Yaskawa INFORM job: A_ROOF_SIDE_0617_2_PAINT_9.JBI

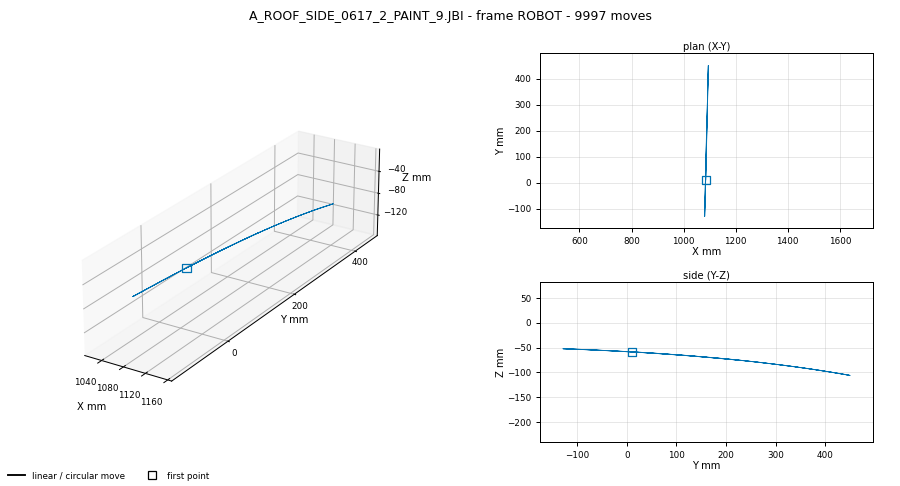
[picture p0: tool path of A_ROOF_SIDE_0617_2_PAINT_9.JBI in frame ROBOT, 9997 of 9997 moves have a stored position in this frame; points joined in program order, loops and branches not executed]
/JOB
//NAME A_ROOF_SIDE_0617_2_PAINT9
//POS
///NPOS 9997,0,0,0,0,0
///TOOL 1
///USER 0
///POSTYPE ROBOT
///RECTAN
///RCONF 1,0,0,0,0,0,0,0,0,0,0,0,0,0,0,0,0,0,0,0,0,0,0,0
C00000=1085.245,10.844,-58.197,174.491,19.105,153.128
C00001=1085.250,11.093,-58.211,174.492,19.107,153.129
C00002=1085.256,11.342,-58.226,174.493,19.109,153.129
C00003=1085.262,11.592,-58.240,174.496,19.111,153.129
C00004=1085.269,11.841,-58.254,174.497,19.113,153.129
C00005=1085.275,12.091,-58.268,174.498,19.115,153.129
C00006=1085.280,12.340,-58.283,174.500,19.118,153.129
C00007=1085.286,12.590,-58.297,174.502,19.119,153.129
C00008=1085.292,12.839,-58.312,174.503,19.121,153.129
C00009=1085.298,13.089,-58.325,174.505,19.123,153.129
C00010=1085.304,13.338,-58.340,174.507,19.125,153.130
C00011=1085.310,13.588,-58.354,174.508,19.127,153.130
C00012=1085.315,13.837,-58.369,174.509,19.129,153.130
C00013=1085.321,14.087,-58.383,174.512,19.131,153.130
C00014=1085.327,14.336,-58.398,174.513,19.133,153.130
C00015=1085.333,14.586,-58.412,174.514,19.134,153.130
C00016=1085.340,14.863,-58.428,174.516,19.137,153.130
C00017=1085.346,15.140,-58.445,174.517,19.139,153.130
C00018=1085.352,15.417,-58.461,174.520,19.141,153.130
C00019=1085.358,15.693,-58.476,174.521,19.143,153.131
C00020=1085.365,15.943,-58.491,174.523,19.145,153.131
C00021=1085.370,16.192,-58.505,174.524,19.147,153.131
C00022=1085.376,16.443,-58.520,174.526,19.149,153.131
C00023=1085.382,16.692,-58.535,174.528,19.151,153.131
C00024=1085.387,16.941,-58.549,174.529,19.153,153.131
C00025=1085.393,17.191,-58.564,174.530,19.155,153.131
C00026=1085.399,17.440,-58.578,174.533,19.157,153.131
C00027=1085.405,17.689,-58.592,174.534,19.159,153.131
C00028=1085.411,17.939,-58.607,174.535,19.161,153.132
C00029=1085.416,18.188,-58.622,174.537,19.163,153.132
C00030=1085.422,18.438,-58.636,174.539,19.165,153.132
C00031=1085.428,18.687,-58.651,174.540,19.167,153.132
C00032=1085.434,18.937,-58.666,174.541,19.168,153.132
C00033=1085.440,19.187,-58.680,174.544,19.171,153.132
C00034=1085.445,19.436,-58.695,174.545,19.173,153.132
C00035=1085.451,19.686,-58.710,174.546,19.174,153.132
C00036=1085.457,19.935,-58.724,174.548,19.177,153.132
C00037=1085.463,20.185,-58.739,174.550,19.178,153.132
C00038=1085.469,20.434,-58.753,174.551,19.181,153.133
C00039=1085.474,20.684,-58.769,174.553,19.183,153.133
C00040=1085.480,20.933,-58.783,174.554,19.185,153.133
C00041=1085.486,21.182,-58.797,174.556,19.186,153.133
C00042=1085.491,21.432,-58.813,174.558,19.189,153.133
C00043=1085.497,21.681,-58.827,174.559,19.191,153.133
C00044=1085.503,21.931,-58.842,174.561,19.192,153.133
C00045=1085.509,22.180,-58.856,174.563,19.195,153.133
C00046=1085.515,22.430,-58.872,174.564,19.196,153.133
C00047=1085.520,22.679,-58.886,174.565,19.198,153.134
C00048=1085.527,22.930,-58.901,174.568,19.200,153.134
C00049=1085.532,23.179,-58.916,174.569,19.202,153.134
C00050=1085.538,23.429,-58.931,174.570,19.204,153.134
C00051=1085.544,23.677,-58.945,174.572,19.206,153.134
C00052=1085.549,23.927,-58.960,174.574,19.208,153.134
C00053=1085.555,24.176,-58.975,174.575,19.210,153.134
C00054=1085.561,24.426,-58.989,174.577,19.212,153.134
C00055=1085.566,24.676,-59.005,174.578,19.214,153.134
C00056=1085.572,24.925,-59.019,174.580,19.216,153.135
C00057=1085.578,25.175,-59.034,174.582,19.218,153.135
C00058=1085.584,25.424,-59.049,174.583,19.220,153.135
C00059=1085.590,25.674,-59.064,174.585,19.222,153.135
C00060=1085.596,25.922,-59.079,174.587,19.224,153.135
C00061=1085.601,26.172,-59.095,174.588,19.226,153.135
C00062=1085.607,26.421,-59.109,174.589,19.228,153.135
C00063=1085.613,26.672,-59.123,174.592,19.230,153.135
C00064=1085.619,26.922,-59.139,174.593,19.232,153.135
C00065=1085.625,27.171,-59.153,174.594,19.233,153.135
C00066=1085.630,27.421,-59.169,174.596,19.236,153.136
C00067=1085.636,27.670,-59.184,174.598,19.237,153.136
C00068=1085.642,27.919,-59.199,174.599,19.239,153.136
C00069=1085.647,28.168,-59.214,174.601,19.241,153.136
C00070=1085.654,28.418,-59.229,174.602,19.243,153.136
C00071=1085.659,28.667,-59.244,174.604,19.245,153.136
C00072=1085.665,28.917,-59.259,174.606,19.247,153.136
C00073=1085.670,29.166,-59.274,174.607,19.249,153.136
C00074=1085.677,29.416,-59.289,174.609,19.251,153.136
C00075=1085.682,29.665,-59.304,174.611,19.253,153.137
C00076=1085.688,29.915,-59.319,174.612,19.255,153.137
C00077=1085.693,30.164,-59.334,174.613,19.257,153.137
C00078=1085.700,30.414,-59.349,174.616,19.259,153.137
C00079=1085.705,30.664,-59.365,174.617,19.261,153.137
C00080=1085.712,30.942,-59.382,174.619,19.263,153.137
C00081=1085.718,31.220,-59.398,174.620,19.265,153.137
C00082=1085.725,31.498,-59.415,174.622,19.268,153.137
C00083=1085.731,31.776,-59.432,174.624,19.270,153.137
C00084=1085.736,32.025,-59.447,174.626,19.272,153.137
C00085=1085.743,32.275,-59.462,174.627,19.274,153.138
C00086=1085.748,32.525,-59.478,174.629,19.276,153.138
C00087=1085.754,32.774,-59.493,174.631,19.278,153.138
C00088=1085.760,33.023,-59.508,174.632,19.279,153.138
C00089=1085.765,33.273,-59.524,174.634,19.282,153.138
C00090=1085.771,33.522,-59.538,174.636,19.283,153.138
C00091=1085.776,33.772,-59.554,174.637,19.285,153.138
C00092=1085.783,34.021,-59.569,174.639,19.287,153.138
C00093=1085.788,34.271,-59.584,174.640,19.289,153.138
C00094=1085.794,34.520,-59.600,174.643,19.291,153.138
C00095=1085.800,34.770,-59.615,174.644,19.293,153.139
C00096=1085.806,35.020,-59.630,174.645,19.295,153.139
C00097=1085.812,35.268,-59.645,174.647,19.298,153.139
C00098=1085.817,35.518,-59.661,174.649,19.299,153.139
C00099=1085.822,35.768,-59.676,174.650,19.301,153.139
C00100=1085.829,36.017,-59.691,174.652,19.303,153.139
C00101=1085.835,36.267,-59.707,174.654,19.305,153.139
C00102=1085.840,36.516,-59.722,174.655,19.307,153.139
C00103=1085.846,36.766,-59.737,174.657,19.309,153.139
C00104=1085.852,37.015,-59.753,174.659,19.311,153.139
C00105=1085.858,37.264,-59.768,174.661,19.313,153.139
C00106=1085.863,37.514,-59.783,174.662,19.315,153.140
C00107=1085.870,37.764,-59.798,174.663,19.316,153.140
C00108=1085.875,38.012,-59.814,174.666,19.319,153.140
C00109=1085.881,38.262,-59.830,174.667,19.320,153.140
C00110=1085.886,38.512,-59.845,174.668,19.322,153.140
C00111=1085.893,38.760,-59.861,174.671,19.324,153.140
C00112=1085.898,39.010,-59.876,174.672,19.326,153.140
C00113=1085.904,39.260,-59.892,174.674,19.328,153.140
C00114=1085.909,39.509,-59.908,174.675,19.330,153.140
C00115=1085.915,39.759,-59.923,174.677,19.332,153.140
C00116=1085.921,40.009,-59.938,174.679,19.334,153.141
C00117=1085.927,40.257,-59.954,174.680,19.336,153.141
C00118=1085.932,40.507,-59.970,174.682,19.338,153.141
C00119=1085.938,40.757,-59.985,174.684,19.340,153.141
C00120=1085.944,41.006,-60.000,174.685,19.342,153.141
C00121=1085.950,41.256,-60.016,174.687,19.344,153.141
C00122=1085.955,41.506,-60.032,174.688,19.346,153.141
C00123=1085.961,41.754,-60.047,174.690,19.348,153.141
C00124=1085.966,42.004,-60.063,174.692,19.350,153.141
C00125=1085.972,42.253,-60.079,174.693,19.352,153.141
C00126=1085.978,42.502,-60.094,174.695,19.354,153.142
C00127=1085.984,42.752,-60.110,174.697,19.356,153.142
C00128=1085.990,43.002,-60.126,174.698,19.357,153.142
C00129=1085.995,43.252,-60.141,174.700,19.360,153.142
C00130=1086.001,43.500,-60.157,174.702,19.361,153.142
C00131=1086.007,43.750,-60.172,174.704,19.364,153.142
C00132=1086.013,43.999,-60.188,174.705,19.365,153.142
C00133=1086.018,44.249,-60.203,174.707,19.367,153.142
C00134=1086.024,44.498,-60.220,174.709,19.369,153.142
C00135=1086.030,44.748,-60.235,174.710,19.371,153.142
C00136=1086.035,44.997,-60.251,174.712,19.373,153.142
C00137=1086.041,45.247,-60.267,174.714,19.375,153.143
C00138=1086.047,45.496,-60.283,174.715,19.377,153.143
C00139=1086.052,45.746,-60.298,174.717,19.379,153.143
C00140=1086.058,45.995,-60.314,174.719,19.381,153.143
C00141=1086.063,46.245,-60.330,174.721,19.383,153.143
C00142=1086.069,46.494,-60.346,174.722,19.385,153.143
C00143=1086.074,46.743,-60.361,174.723,19.387,153.143
C00144=1086.081,47.022,-60.379,174.726,19.389,153.143
C00145=1086.087,47.300,-60.397,174.728,19.391,153.143
C00146=1086.092,47.578,-60.415,174.729,19.393,153.144
C00147=1086.100,47.857,-60.432,174.731,19.396,153.144
C00148=1086.105,48.105,-60.448,174.733,19.398,153.144
C00149=1086.111,48.355,-60.465,174.735,19.400,153.144
C00150=1086.117,48.605,-60.480,174.736,19.402,153.144
C00151=1086.123,48.854,-60.496,174.738,19.404,153.144
C00152=1086.127,49.103,-60.513,174.740,19.406,153.144
C00153=1086.133,49.353,-60.528,174.742,19.408,153.144
C00154=1086.139,49.602,-60.545,174.743,19.410,153.144
C00155=1086.144,49.852,-60.560,174.745,19.411,153.144
C00156=1086.150,50.102,-60.576,174.747,19.413,153.144
C00157=1086.156,50.350,-60.592,174.748,19.415,153.145
C00158=1086.161,50.600,-60.608,174.750,19.417,153.145
C00159=1086.167,50.850,-60.624,174.752,19.419,153.145
C00160=1086.173,51.099,-60.640,174.753,19.421,153.145
C00161=1086.179,51.348,-60.657,174.755,19.423,153.145
C00162=1086.184,51.598,-60.672,174.757,19.425,153.145
C00163=1086.190,51.847,-60.688,174.759,19.427,153.145
C00164=1086.196,52.096,-60.704,174.760,19.429,153.145
C00165=1086.202,52.346,-60.721,174.762,19.431,153.145
C00166=1086.207,52.596,-60.737,174.764,19.433,153.145
C00167=1086.212,52.845,-60.753,174.765,19.434,153.145
C00168=1086.218,53.094,-60.769,174.767,19.436,153.145
C00169=1086.224,53.343,-60.785,174.769,19.438,153.146
C00170=1086.230,53.593,-60.801,174.771,19.440,153.146
C00171=1086.236,53.843,-60.817,174.772,19.442,153.146
C00172=1086.242,54.092,-60.833,174.774,19.444,153.146
C00173=1086.248,54.341,-60.849,174.776,19.446,153.146
C00174=1086.253,54.590,-60.865,174.777,19.447,153.146
C00175=1086.258,54.840,-60.881,174.779,19.450,153.146
C00176=1086.264,55.089,-60.898,174.781,19.451,153.146
C00177=1086.270,55.339,-60.914,174.783,19.454,153.146
C00178=1086.276,55.588,-60.930,174.784,19.455,153.146
C00179=1086.282,55.838,-60.946,174.787,19.457,153.146
C00180=1086.288,56.087,-60.963,174.788,19.460,153.146
C00181=1086.293,56.337,-60.978,174.789,19.461,153.146
C00182=1086.299,56.587,-60.995,174.792,19.463,153.146
C00183=1086.305,56.836,-61.011,174.793,19.465,153.146
C00184=1086.310,57.085,-61.027,174.795,19.467,153.147
C00185=1086.316,57.334,-61.044,174.797,19.469,153.147
C00186=1086.322,57.583,-61.060,174.799,19.471,153.147
C00187=1086.328,57.833,-61.076,174.800,19.473,153.147
C00188=1086.333,58.082,-61.093,174.802,19.474,153.147
C00189=1086.339,58.332,-61.109,174.804,19.476,153.147
C00190=1086.345,58.581,-61.125,174.805,19.478,153.147
C00191=1086.351,58.830,-61.142,174.808,19.480,153.147
C00192=1086.357,59.080,-61.158,174.809,19.482,153.147
C00193=1086.362,59.329,-61.175,174.811,19.484,153.147
C00194=1086.368,59.579,-61.191,174.813,19.486,153.147
C00195=1086.374,59.828,-61.207,174.814,19.487,153.147
C00196=1086.380,60.077,-61.224,174.816,19.489,153.147
C00197=1086.386,60.327,-61.240,174.818,19.491,153.147
C00198=1086.391,60.576,-61.257,174.820,19.493,153.148
C00199=1086.397,60.826,-61.273,174.821,19.495,153.148
C00200=1086.403,61.075,-61.289,174.824,19.497,153.148
C00201=1086.409,61.324,-61.305,174.825,19.498,153.148
C00202=1086.415,61.574,-61.322,174.827,19.501,153.148
C00203=1086.420,61.823,-61.339,174.829,19.502,153.148
C00204=1086.426,62.073,-61.355,174.830,19.504,153.148
C00205=1086.432,62.322,-61.371,174.832,19.506,153.148
C00206=1086.438,62.571,-61.387,174.834,19.507,153.148
C00207=1086.443,62.821,-61.404,174.836,19.510,153.148
C00208=1086.451,63.099,-61.422,174.838,19.512,153.148
C00209=1086.457,63.376,-61.441,174.840,19.513,153.148
C00210=1086.463,63.655,-61.459,174.842,19.516,153.148
C00211=1086.470,63.933,-61.477,174.844,19.518,153.148
C00212=1086.476,64.182,-61.494,174.845,19.519,153.148
C00213=1086.481,64.432,-61.511,174.848,19.521,153.148
C00214=1086.487,64.681,-61.527,174.849,19.523,153.149
C00215=1086.492,64.930,-61.544,174.851,19.525,153.149
C00216=1086.498,65.180,-61.561,174.853,19.527,153.149
C00217=1086.504,65.429,-61.577,174.855,19.529,153.149
C00218=1086.509,65.679,-61.594,174.856,19.531,153.149
C00219=1086.515,65.928,-61.610,174.858,19.532,153.149
C00220=1086.521,66.177,-61.628,174.860,19.534,153.149
C00221=1086.527,66.426,-61.644,174.862,19.536,153.149
C00222=1086.532,66.676,-61.661,174.864,19.538,153.149
C00223=1086.538,66.925,-61.677,174.865,19.540,153.149
C00224=1086.544,67.175,-61.693,174.867,19.542,153.149
C00225=1086.550,67.424,-61.711,174.869,19.543,153.149
C00226=1086.556,67.674,-61.727,174.871,19.545,153.149
C00227=1086.561,67.923,-61.744,174.872,19.547,153.149
C00228=1086.567,68.173,-61.760,174.875,19.549,153.149
C00229=1086.573,68.422,-61.778,174.876,19.551,153.149
C00230=1086.579,68.671,-61.794,174.878,19.553,153.149
C00231=1086.584,68.921,-61.811,174.880,19.554,153.149
C00232=1086.590,69.170,-61.828,174.882,19.557,153.150
C00233=1086.595,69.419,-61.845,174.883,19.558,153.150
C00234=1086.601,69.669,-61.861,174.885,19.560,153.150
C00235=1086.607,69.918,-61.879,174.887,19.562,153.150
C00236=1086.612,70.167,-61.896,174.889,19.564,153.150
C00237=1086.618,70.417,-61.912,174.891,19.566,153.150
C00238=1086.624,70.666,-61.929,174.892,19.568,153.150
C00239=1086.629,70.915,-61.946,174.895,19.570,153.150
C00240=1086.635,71.165,-61.963,174.896,19.571,153.150
C00241=1086.641,71.414,-61.980,174.898,19.573,153.150
C00242=1086.647,71.664,-61.997,174.900,19.575,153.150
C00243=1086.652,71.913,-62.014,174.902,19.577,153.150
C00244=1086.658,72.162,-62.031,174.903,19.579,153.150
C00245=1086.663,72.412,-62.047,174.906,19.581,153.150
C00246=1086.669,72.661,-62.065,174.907,19.582,153.150
C00247=1086.675,72.910,-62.081,174.909,19.585,153.150
C00248=1086.680,73.159,-62.099,174.911,19.586,153.150
C00249=1086.686,73.409,-62.116,174.913,19.588,153.150
C00250=1086.692,73.658,-62.133,174.914,19.590,153.151
C00251=1086.698,73.908,-62.150,174.917,19.592,153.151
C00252=1086.703,74.158,-62.167,174.918,19.593,153.151
C00253=1086.709,74.406,-62.184,174.921,19.595,153.151
C00254=1086.714,74.656,-62.201,174.922,19.597,153.151
C00255=1086.720,74.905,-62.218,174.924,19.599,153.151
C00256=1086.726,75.154,-62.234,174.926,19.601,153.151
C00257=1086.732,75.404,-62.252,174.928,19.603,153.151
C00258=1086.737,75.654,-62.269,174.929,19.604,153.151
C00259=1086.743,75.902,-62.286,174.932,19.606,153.151
C00260=1086.749,76.152,-62.304,174.933,19.608,153.151
C00261=1086.754,76.401,-62.321,174.935,19.610,153.151
C00262=1086.760,76.650,-62.337,174.937,19.612,153.151
C00263=1086.766,76.900,-62.355,174.939,19.614,153.151
C00264=1086.772,77.149,-62.372,174.940,19.615,153.151
C00265=1086.777,77.399,-62.389,174.943,19.617,153.151
C00266=1086.783,77.648,-62.406,174.944,19.619,153.151
C00267=1086.789,77.897,-62.424,174.947,19.621,153.151
C00268=1086.795,78.147,-62.441,174.948,19.622,153.151
C00269=1086.800,78.396,-62.458,174.950,19.624,153.151
C00270=1086.806,78.646,-62.475,174.952,19.626,153.151
C00271=1086.812,78.895,-62.492,174.954,19.628,153.151
C00272=1086.818,79.173,-62.512,174.956,19.630,153.151
C00273=1086.824,79.450,-62.531,174.958,19.632,153.152
C00274=1086.830,79.728,-62.550,174.960,19.634,153.152
C00275=1086.836,80.007,-62.570,174.962,19.636,153.152
C00276=1086.843,80.256,-62.587,174.964,19.637,153.152
C00277=1086.848,80.505,-62.604,174.966,19.640,153.152
C00278=1086.853,80.754,-62.621,174.967,19.641,153.152
C00279=1086.859,81.003,-62.639,174.970,19.643,153.152
C00280=1086.865,81.253,-62.657,174.972,19.645,153.152
C00281=1086.870,81.503,-62.673,174.973,19.647,153.152
C00282=1086.876,81.752,-62.691,174.976,19.649,153.152
C00283=1086.881,82.001,-62.709,174.977,19.650,153.152
C00284=1086.887,82.251,-62.727,174.979,19.652,153.152
C00285=1086.893,82.500,-62.743,174.981,19.654,153.152
C00286=1086.898,82.749,-62.761,174.983,19.656,153.152
C00287=1086.904,82.998,-62.778,174.985,19.657,153.152
C00288=1086.910,83.247,-62.795,174.987,19.659,153.152
C00289=1086.916,83.497,-62.813,174.988,19.661,153.152
C00290=1086.921,83.747,-62.830,174.991,19.663,153.152
C00291=1086.927,83.996,-62.848,174.992,19.665,153.152
C00292=1086.933,84.245,-62.866,174.994,19.667,153.152
C00293=1086.938,84.494,-62.883,174.996,19.668,153.152
C00294=1086.944,84.743,-62.901,174.998,19.670,153.152
C00295=1086.949,84.992,-62.918,175.000,19.672,153.152
C00296=1086.955,85.243,-62.936,175.002,19.674,153.152
C00297=1086.961,85.492,-62.953,175.003,19.675,153.152
C00298=1086.966,85.741,-62.971,175.006,19.677,153.152
C00299=1086.972,85.990,-62.988,175.007,19.679,153.152
C00300=1086.978,86.240,-63.006,175.009,19.681,153.152
C00301=1086.983,86.489,-63.024,175.012,19.683,153.152
C00302=1086.989,86.738,-63.041,175.013,19.684,153.153
C00303=1086.995,86.987,-63.059,175.016,19.686,153.152
C00304=1087.000,87.237,-63.076,175.017,19.687,153.152
C00305=1087.006,87.486,-63.094,175.020,19.689,153.152
C00306=1087.012,87.736,-63.112,175.021,19.691,153.153
C00307=1087.017,87.985,-63.129,175.023,19.693,153.153
C00308=1087.023,88.234,-63.147,175.025,19.694,153.153
C00309=1087.029,88.484,-63.165,175.027,19.696,153.153
C00310=1087.035,88.733,-63.182,175.029,19.698,153.153
C00311=1087.040,88.982,-63.200,175.031,19.700,153.153
C00312=1087.046,89.232,-63.218,175.032,19.701,153.153
C00313=1087.052,89.481,-63.235,175.035,19.703,153.153
C00314=1087.058,89.730,-63.253,175.037,19.705,153.153
C00315=1087.063,89.979,-63.271,175.039,19.707,153.153
C00316=1087.069,90.228,-63.288,175.041,19.708,153.153
C00317=1087.075,90.478,-63.306,175.043,19.710,153.153
C00318=1087.080,90.727,-63.324,175.045,19.712,153.153
C00319=1087.087,90.977,-63.342,175.046,19.713,153.153
C00320=1087.092,91.226,-63.359,175.049,19.715,153.153
C00321=1087.097,91.475,-63.378,175.050,19.717,153.153
C00322=1087.103,91.724,-63.396,175.052,19.719,153.153
C00323=1087.109,91.973,-63.414,175.055,19.721,153.153
C00324=1087.114,92.223,-63.431,175.056,19.722,153.153
C00325=1087.120,92.472,-63.449,175.059,19.724,153.153
C00326=1087.125,92.722,-63.468,175.060,19.726,153.153
C00327=1087.131,92.971,-63.485,175.062,19.728,153.153
C00328=1087.137,93.220,-63.503,175.064,19.729,153.153
C00329=1087.142,93.469,-63.521,175.066,19.731,153.153
C00330=1087.148,93.718,-63.539,175.068,19.732,153.153
C00331=1087.154,93.968,-63.557,175.070,19.734,153.153
C00332=1087.159,94.217,-63.575,175.072,19.736,153.153
C00333=1087.165,94.467,-63.593,175.074,19.738,153.153
C00334=1087.170,94.716,-63.611,175.076,19.740,153.153
C00335=1087.176,94.965,-63.629,175.078,19.741,153.153
C00336=1087.182,95.243,-63.649,175.080,19.743,153.153
C00337=1087.188,95.521,-63.669,175.082,19.745,153.153
C00338=1087.195,95.799,-63.689,175.085,19.747,153.153
C00339=1087.202,96.077,-63.710,175.087,19.749,153.153
C00340=1087.206,96.327,-63.728,175.088,19.751,153.153
C00341=1087.212,96.576,-63.745,175.091,19.752,153.153
C00342=1087.218,96.825,-63.764,175.092,19.754,153.153
C00343=1087.224,97.074,-63.781,175.095,19.756,153.153
C00344=1087.229,97.324,-63.800,175.097,19.758,153.153
C00345=1087.235,97.572,-63.818,175.099,19.759,153.153
C00346=1087.241,97.822,-63.836,175.101,19.761,153.153
C00347=1087.246,98.071,-63.854,175.103,19.762,153.153
C00348=1087.252,98.321,-63.873,175.105,19.764,153.153
C00349=1087.258,98.570,-63.891,175.107,19.766,153.153
C00350=1087.263,98.820,-63.909,175.109,19.768,153.153
C00351=1087.269,99.068,-63.927,175.111,19.769,153.153
C00352=1087.275,99.318,-63.945,175.113,19.771,153.153
C00353=1087.281,99.567,-63.963,175.115,19.773,153.153
C00354=1087.287,99.816,-63.982,175.117,19.774,153.153
C00355=1087.292,100.065,-64.000,175.119,19.776,153.153
C00356=1087.298,100.315,-64.018,175.121,19.778,153.153
C00357=1087.303,100.564,-64.037,175.123,19.779,153.153
C00358=1087.309,100.814,-64.054,175.125,19.781,153.153
C00359=1087.314,101.062,-64.073,175.127,19.782,153.153
C00360=1087.321,101.312,-64.091,175.129,19.784,153.153
C00361=1087.326,101.561,-64.109,175.132,19.786,153.153
C00362=1087.332,101.811,-64.128,175.133,19.788,153.153
C00363=1087.337,102.060,-64.146,175.135,19.790,153.153
C00364=1087.343,102.309,-64.165,175.137,19.791,153.153
C00365=1087.349,102.558,-64.182,175.139,19.793,153.153
C00366=1087.354,102.807,-64.202,175.142,19.795,153.153
C00367=1087.360,103.057,-64.219,175.143,19.796,153.153
C00368=1087.365,103.306,-64.239,175.145,19.798,153.153
C00369=1087.371,103.555,-64.256,175.147,19.799,153.153
C00370=1087.377,103.804,-64.275,175.150,19.801,153.153
C00371=1087.381,104.054,-64.293,175.152,19.803,153.153
C00372=1087.388,104.303,-64.312,175.153,19.804,153.153
C00373=1087.393,104.552,-64.330,175.156,19.806,153.153
C00374=1087.399,104.801,-64.349,175.157,19.807,153.153
C00375=1087.404,105.051,-64.367,175.160,19.809,153.153
C00376=1087.410,105.300,-64.386,175.162,19.811,153.153
C00377=1087.416,105.549,-64.405,175.164,19.812,153.153
C00378=1087.421,105.798,-64.423,175.166,19.814,153.153
C00379=1087.427,106.048,-64.442,175.167,19.816,153.153
C00380=1087.432,106.297,-64.460,175.170,19.817,153.153
C00381=1087.438,106.546,-64.479,175.172,19.819,153.153
C00382=1087.444,106.796,-64.498,175.174,19.821,153.153
C00383=1087.450,107.045,-64.515,175.176,19.822,153.153
C00384=1087.455,107.294,-64.535,175.178,19.824,153.153
C00385=1087.461,107.543,-64.552,175.180,19.826,153.153
C00386=1087.466,107.793,-64.571,175.183,19.827,153.153
C00387=1087.472,108.042,-64.591,175.184,19.829,153.153
C00388=1087.478,108.291,-64.608,175.187,19.831,153.153
C00389=1087.483,108.540,-64.628,175.189,19.832,153.152
C00390=1087.489,108.789,-64.646,175.191,19.834,153.153
C00391=1087.495,109.038,-64.665,175.193,19.836,153.153
C00392=1087.500,109.288,-64.684,175.195,19.837,153.152
C00393=1087.506,109.537,-64.702,175.197,19.839,153.152
C00394=1087.512,109.786,-64.721,175.199,19.840,153.152
C00395=1087.518,110.036,-64.739,175.201,19.842,153.152
C00396=1087.523,110.285,-64.758,175.203,19.844,153.152
C00397=1087.529,110.534,-64.777,175.206,19.845,153.152
C00398=1087.535,110.783,-64.796,175.207,19.847,153.152
C00399=1087.540,111.033,-64.814,175.210,19.848,153.152
C00400=1087.546,111.311,-64.836,175.212,19.850,153.152
C00401=1087.553,111.589,-64.856,175.215,19.852,153.152
C00402=1087.559,111.866,-64.877,175.217,19.854,153.152
C00403=1087.566,112.145,-64.898,175.219,19.856,153.152
C00404=1087.571,112.394,-64.917,175.221,19.857,153.152
C00405=1087.577,112.643,-64.936,175.223,19.859,153.152
C00406=1087.582,112.893,-64.955,175.225,19.860,153.152
C00407=1087.588,113.141,-64.974,175.227,19.862,153.152
C00408=1087.594,113.390,-64.993,175.230,19.864,153.152
C00409=1087.599,113.640,-65.011,175.231,19.865,153.152
C00410=1087.605,113.890,-65.031,175.234,19.867,153.152
C00411=1087.611,114.138,-65.049,175.236,19.869,153.152
C00412=1087.616,114.388,-65.068,175.238,19.870,153.152
C00413=1087.622,114.637,-65.087,175.240,19.872,153.152
C00414=1087.627,114.886,-65.106,175.243,19.873,153.152
C00415=1087.633,115.135,-65.125,175.244,19.875,153.152
C00416=1087.638,115.385,-65.145,175.247,19.877,153.152
C00417=1087.644,115.634,-65.164,175.249,19.878,153.152
C00418=1087.649,115.883,-65.183,175.251,19.880,153.152
C00419=1087.655,116.132,-65.202,175.253,19.882,153.152
C00420=1087.660,116.381,-65.221,175.255,19.883,153.152
C00421=1087.666,116.631,-65.240,175.257,19.885,153.152
C00422=1087.671,116.880,-65.259,175.259,19.886,153.151
C00423=1087.676,117.129,-65.278,175.262,19.888,153.151
C00424=1087.682,117.378,-65.298,175.263,19.890,153.152
C00425=1087.689,117.627,-65.316,175.266,19.891,153.151
C00426=1087.694,117.876,-65.335,175.268,19.893,153.151
C00427=1087.699,118.125,-65.354,175.270,19.894,153.151
C00428=1087.705,118.375,-65.374,175.272,19.896,153.151
C00429=1087.711,118.624,-65.393,175.275,19.897,153.151
C00430=1087.716,118.873,-65.412,175.276,19.899,153.151
C00431=1087.721,119.122,-65.431,175.279,19.900,153.151
C00432=1087.727,119.372,-65.450,175.281,19.902,153.151
C00433=1087.733,119.621,-65.469,175.283,19.903,153.151
C00434=1087.738,119.870,-65.488,175.285,19.905,153.151
C00435=1087.744,120.120,-65.508,175.288,19.907,153.151
C00436=1087.749,120.369,-65.527,175.289,19.908,153.151
C00437=1087.755,120.618,-65.546,175.292,19.910,153.151
C00438=1087.760,120.866,-65.566,175.294,19.912,153.151
C00439=1087.766,121.116,-65.585,175.296,19.913,153.151
C00440=1087.772,121.365,-65.604,175.298,19.915,153.151
C00441=1087.777,121.615,-65.623,175.301,19.916,153.151
C00442=1087.782,121.864,-65.643,175.302,19.918,153.151
C00443=1087.788,122.113,-65.662,175.305,19.919,153.151
C00444=1087.793,122.362,-65.682,175.307,19.921,153.151
C00445=1087.799,122.612,-65.701,175.309,19.922,153.151
C00446=1087.805,122.861,-65.720,175.311,19.924,153.151
C00447=1087.811,123.110,-65.740,175.314,19.926,153.150
C00448=1087.816,123.358,-65.759,175.315,19.927,153.150
C00449=1087.822,123.608,-65.779,175.318,19.929,153.150
C00450=1087.827,123.857,-65.798,175.320,19.930,153.150
C00451=1087.833,124.107,-65.817,175.322,19.932,153.150
C00452=1087.839,124.356,-65.837,175.324,19.933,153.150
C00453=1087.845,124.605,-65.856,175.327,19.935,153.150
C00454=1087.850,124.854,-65.875,175.329,19.937,153.150
C00455=1087.855,125.103,-65.894,175.331,19.938,153.150
C00456=1087.861,125.352,-65.914,175.333,19.940,153.150
C00457=1087.867,125.601,-65.934,175.336,19.941,153.150
C00458=1087.872,125.851,-65.953,175.337,19.942,153.150
C00459=1087.878,126.100,-65.973,175.340,19.944,153.150
C00460=1087.884,126.349,-65.993,175.342,19.946,153.150
C00461=1087.889,126.599,-66.012,175.344,19.947,153.150
C00462=1087.895,126.848,-66.032,175.346,19.949,153.150
C00463=1087.901,127.096,-66.051,175.349,19.950,153.149
C00464=1087.907,127.375,-66.073,175.351,19.952,153.149
C00465=1087.914,127.653,-66.094,175.354,19.954,153.149
C00466=1087.920,127.930,-66.116,175.356,19.955,153.149
C00467=1087.926,128.208,-66.138,175.359,19.957,153.149
C00468=1087.931,128.458,-66.158,175.361,19.959,153.149
C00469=1087.937,128.707,-66.178,175.363,19.960,153.149
C00470=1087.943,128.956,-66.197,175.365,19.961,153.149
C00471=1087.949,129.206,-66.217,175.368,19.963,153.149
C00472=1087.955,129.454,-66.237,175.369,19.964,153.149
C00473=1087.960,129.704,-66.256,175.372,19.965,153.149
C00474=1087.966,129.953,-66.276,175.375,19.967,153.149
C00475=1087.971,130.202,-66.296,175.377,19.968,153.148
C00476=1087.977,130.451,-66.316,175.379,19.970,153.148
C00477=1087.983,130.701,-66.335,175.381,19.971,153.148
C00478=1087.989,130.950,-66.355,175.384,19.973,153.148
C00479=1087.995,131.199,-66.374,175.385,19.974,153.148
C00480=1088.000,131.448,-66.395,175.388,19.975,153.148
C00481=1088.006,131.697,-66.415,175.390,19.977,153.148
C00482=1088.012,131.946,-66.434,175.393,19.979,153.148
C00483=1088.018,132.195,-66.454,175.395,19.980,153.148
C00484=1088.023,132.445,-66.473,175.397,19.981,153.148
C00485=1088.029,132.694,-66.494,175.400,19.983,153.148
C00486=1088.034,132.943,-66.513,175.401,19.984,153.148
C00487=1088.040,133.192,-66.533,175.404,19.986,153.147
C00488=1088.046,133.441,-66.553,175.406,19.987,153.147
C00489=1088.051,133.690,-66.573,175.409,19.989,153.147
C00490=1088.057,133.940,-66.593,175.410,19.990,153.147
C00491=1088.063,134.188,-66.613,175.413,19.992,153.147
C00492=1088.067,134.438,-66.633,175.416,19.993,153.147
C00493=1088.073,134.687,-66.653,175.418,19.995,153.147
C00494=1088.079,134.936,-66.673,175.420,19.996,153.147
C00495=1088.084,135.186,-66.693,175.422,19.998,153.147
C00496=1088.090,135.434,-66.713,175.425,19.999,153.147
C00497=1088.096,135.683,-66.733,175.427,20.001,153.147
C00498=1088.101,135.933,-66.752,175.429,20.002,153.147
C00499=1088.107,136.182,-66.772,175.431,20.004,153.146
C00500=1088.113,136.431,-66.793,175.434,20.005,153.146
C00501=1088.119,136.680,-66.813,175.436,20.007,153.146
C00502=1088.124,136.929,-66.833,175.438,20.008,153.146
C00503=1088.130,137.178,-66.853,175.440,20.010,153.146
C00504=1088.135,137.427,-66.873,175.443,20.011,153.146
C00505=1088.141,137.676,-66.893,175.446,20.013,153.146
C00506=1088.146,137.926,-66.912,175.447,20.014,153.146
C00507=1088.152,138.175,-66.933,175.450,20.015,153.146
C00508=1088.158,138.424,-66.953,175.452,20.017,153.146
C00509=1088.163,138.673,-66.973,175.455,20.019,153.146
C00510=1088.169,138.921,-66.993,175.456,20.020,153.146
C00511=1088.174,139.171,-67.014,175.459,20.021,153.145
C00512=1088.180,139.420,-67.033,175.462,20.022,153.145
C00513=1088.185,139.669,-67.054,175.464,20.024,153.145
C00514=1088.190,139.918,-67.074,175.466,20.025,153.145
C00515=1088.197,140.168,-67.095,175.468,20.026,153.145
C00516=1088.202,140.417,-67.115,175.471,20.028,153.145
C00517=1088.208,140.666,-67.135,175.473,20.030,153.145
C00518=1088.214,140.915,-67.156,175.475,20.031,153.145
C00519=1088.220,141.164,-67.176,175.478,20.032,153.145
C00520=1088.225,141.413,-67.196,175.480,20.034,153.144
C00521=1088.230,141.663,-67.216,175.483,20.035,153.144
C00522=1088.236,141.911,-67.236,175.485,20.037,153.144
C00523=1088.241,142.160,-67.257,175.487,20.038,153.144
C00524=1088.246,142.410,-67.277,175.489,20.040,153.144
C00525=1088.253,142.659,-67.297,175.492,20.041,153.144
C00526=1088.258,142.908,-67.318,175.494,20.043,153.144
C00527=1088.263,143.157,-67.339,175.496,20.044,153.144
C00528=1088.270,143.435,-67.361,175.499,20.046,153.144
C00529=1088.276,143.713,-67.384,175.502,20.047,153.144
C00530=1088.282,143.990,-67.407,175.505,20.049,153.143
C00531=1088.289,144.268,-67.430,175.507,20.050,153.143
C00532=1088.295,144.518,-67.450,175.510,20.052,153.143
C00533=1088.300,144.767,-67.471,175.511,20.053,153.143
C00534=1088.306,145.016,-67.491,175.514,20.055,153.143
C00535=1088.311,145.265,-67.511,175.516,20.056,153.143
C00536=1088.316,145.514,-67.532,175.519,20.058,153.143
C00537=1088.322,145.763,-67.552,175.521,20.059,153.143
C00538=1088.328,146.013,-67.573,175.523,20.060,153.143
C00539=1088.333,146.262,-67.593,175.526,20.062,153.143
C00540=1088.339,146.511,-67.614,175.528,20.063,153.142
C00541=1088.345,146.759,-67.635,175.531,20.065,153.142
C00542=1088.350,147.008,-67.655,175.533,20.066,153.142
C00543=1088.356,147.258,-67.676,175.535,20.067,153.142
C00544=1088.362,147.507,-67.696,175.538,20.069,153.142
C00545=1088.367,147.756,-67.717,175.540,20.070,153.142
C00546=1088.373,148.005,-67.737,175.543,20.072,153.142
C00547=1088.378,148.254,-67.759,175.545,20.073,153.142
C00548=1088.385,148.503,-67.779,175.547,20.074,153.141
C00549=1088.390,148.752,-67.799,175.550,20.075,153.141
C00550=1088.395,149.001,-67.820,175.552,20.077,153.141
C00551=1088.401,149.250,-67.841,175.555,20.078,153.141
C00552=1088.406,149.499,-67.862,175.557,20.080,153.141
C00553=1088.412,149.749,-67.883,175.560,20.081,153.141
C00554=1088.417,149.998,-67.903,175.562,20.082,153.141
C00555=1088.424,150.246,-67.924,175.564,20.084,153.141
C00556=1088.429,150.495,-67.944,175.567,20.085,153.141
C00557=1088.435,150.745,-67.965,175.569,20.087,153.140
C00558=1088.440,150.994,-67.986,175.572,20.088,153.140
C00559=1088.445,151.243,-68.007,175.574,20.089,153.140
C00560=1088.451,151.492,-68.028,175.576,20.091,153.140
C00561=1088.457,151.742,-68.049,175.579,20.092,153.140
C00562=1088.462,151.990,-68.070,175.581,20.094,153.140
C00563=1088.467,152.239,-68.091,175.584,20.095,153.140
C00564=1088.473,152.488,-68.111,175.587,20.096,153.139
C00565=1088.480,152.737,-68.132,175.588,20.097,153.139
C00566=1088.485,152.986,-68.153,175.591,20.099,153.139
C00567=1088.490,153.235,-68.174,175.593,20.100,153.139
C00568=1088.496,153.485,-68.195,175.596,20.102,153.139
C00569=1088.501,153.734,-68.215,175.599,20.103,153.139
C00570=1088.507,153.982,-68.237,175.601,20.105,153.139
C00571=1088.512,154.231,-68.257,175.603,20.106,153.139
C00572=1088.518,154.481,-68.279,175.605,20.107,153.139
C00573=1088.524,154.730,-68.299,175.608,20.109,153.138
C00574=1088.529,154.978,-68.321,175.610,20.110,153.138
C00575=1088.535,155.228,-68.342,175.613,20.112,153.138
C00576=1088.541,155.477,-68.363,175.616,20.113,153.138
C00577=1088.546,155.726,-68.383,175.618,20.114,153.138
C00578=1088.552,155.975,-68.405,175.620,20.115,153.138
C00579=1088.557,156.224,-68.426,175.623,20.117,153.138
C00580=1088.563,156.473,-68.447,175.625,20.118,153.138
C00581=1088.569,156.722,-68.468,175.628,20.120,153.137
C00582=1088.574,156.971,-68.489,175.630,20.121,153.137
C00583=1088.579,157.220,-68.510,175.633,20.123,153.137
C00584=1088.585,157.470,-68.532,175.635,20.124,153.137
C00585=1088.590,157.719,-68.552,175.637,20.125,153.137
C00586=1088.596,157.967,-68.574,175.640,20.126,153.137
C00587=1088.602,158.216,-68.595,175.643,20.128,153.137
C00588=1088.607,158.466,-68.616,175.645,20.129,153.136
C00589=1088.613,158.715,-68.638,175.648,20.130,153.136
C00590=1088.619,158.963,-68.659,175.650,20.132,153.136
C00591=1088.624,159.212,-68.679,175.653,20.133,153.136
C00592=1088.631,159.490,-68.703,175.656,20.134,153.136
C00593=1088.636,159.768,-68.727,175.658,20.136,153.136
C00594=1088.643,160.046,-68.751,175.661,20.137,153.136
C00595=1088.649,160.323,-68.775,175.663,20.139,153.135
C00596=1088.655,160.573,-68.795,175.666,20.140,153.135
C00597=1088.660,160.821,-68.817,175.669,20.141,153.135
C00598=1088.666,161.070,-68.838,175.671,20.143,153.135
C00599=1088.671,161.319,-68.860,175.674,20.144,153.135
C00600=1088.677,161.569,-68.881,175.676,20.146,153.135
C00601=1088.683,161.817,-68.902,175.679,20.147,153.134
C00602=1088.688,162.066,-68.924,175.681,20.148,153.134
C00603=1088.694,162.315,-68.946,175.683,20.149,153.134
C00604=1088.699,162.565,-68.967,175.686,20.151,153.134
C00605=1088.704,162.814,-68.989,175.688,20.152,153.134
C00606=1088.710,163.063,-69.010,175.691,20.154,153.134
C00607=1088.716,163.311,-69.031,175.694,20.155,153.134
C00608=1088.721,163.561,-69.054,175.696,20.157,153.134
C00609=1088.726,163.810,-69.074,175.699,20.158,153.134
C00610=1088.731,164.058,-69.096,175.701,20.160,153.133
C00611=1088.737,164.308,-69.118,175.704,20.161,153.133
C00612=1088.742,164.557,-69.139,175.706,20.162,153.133
C00613=1088.748,164.806,-69.161,175.708,20.163,153.133
C00614=1088.754,165.054,-69.182,175.711,20.165,153.133
C00615=1088.759,165.303,-69.204,175.713,20.166,153.133
C00616=1088.764,165.553,-69.225,175.716,20.168,153.133
C00617=1088.769,165.802,-69.247,175.719,20.169,153.132
C00618=1088.775,166.051,-69.269,175.721,20.170,153.132
C00619=1088.780,166.300,-69.290,175.724,20.172,153.132
C00620=1088.786,166.549,-69.312,175.727,20.173,153.132
C00621=1088.791,166.798,-69.334,175.729,20.175,153.132
C00622=1088.797,167.047,-69.356,175.732,20.176,153.132
C00623=1088.803,167.295,-69.377,175.734,20.177,153.132
C00624=1088.808,167.544,-69.399,175.736,20.178,153.131
C00625=1088.814,167.793,-69.420,175.739,20.180,153.131
C00626=1088.819,168.042,-69.442,175.741,20.181,153.131
C00627=1088.825,168.291,-69.464,175.744,20.182,153.131
C00628=1088.830,168.540,-69.486,175.747,20.183,153.131
C00629=1088.836,168.789,-69.507,175.749,20.185,153.131
C00630=1088.841,169.038,-69.529,175.752,20.186,153.131
C00631=1088.847,169.288,-69.551,175.754,20.188,153.130
C00632=1088.852,169.536,-69.573,175.757,20.189,153.130
C00633=1088.858,169.786,-69.594,175.760,20.190,153.130
C00634=1088.863,170.035,-69.617,175.762,20.192,153.130
C00635=1088.869,170.284,-69.638,175.765,20.193,153.130
C00636=1088.875,170.532,-69.661,175.768,20.194,153.130
C00637=1088.879,170.781,-69.683,175.769,20.195,153.129
C00638=1088.886,171.030,-69.704,175.772,20.197,153.129
C00639=1088.890,171.279,-69.726,175.775,20.198,153.129
C00640=1088.897,171.528,-69.748,175.777,20.199,153.129
C00641=1088.901,171.777,-69.770,175.780,20.201,153.129
C00642=1088.908,172.027,-69.791,175.783,20.202,153.129
C00643=1088.913,172.275,-69.814,175.785,20.203,153.129
C00644=1088.919,172.524,-69.836,175.788,20.205,153.128
C00645=1088.924,172.773,-69.858,175.790,20.206,153.128
C00646=1088.930,173.022,-69.879,175.793,20.207,153.128
C00647=1088.935,173.271,-69.901,175.796,20.209,153.128
C00648=1088.941,173.520,-69.924,175.798,20.210,153.128
C00649=1088.947,173.769,-69.945,175.801,20.211,153.128
C00650=1088.952,174.018,-69.968,175.803,20.213,153.127
C00651=1088.958,174.267,-69.989,175.806,20.214,153.127
C00652=1088.963,174.516,-70.012,175.809,20.215,153.127
C00653=1088.969,174.765,-70.034,175.812,20.216,153.127
C00654=1088.974,175.014,-70.055,175.814,20.218,153.127
C00655=1088.980,175.263,-70.078,175.817,20.219,153.127
C00656=1088.986,175.540,-70.102,175.820,20.220,153.126
C00657=1088.992,175.817,-70.127,175.822,20.222,153.126
C00658=1088.998,176.095,-70.152,175.825,20.223,153.126
C00659=1089.005,176.372,-70.177,175.828,20.225,153.126
C00660=1089.010,176.621,-70.199,175.831,20.226,153.125
C00661=1089.017,176.870,-70.221,175.834,20.227,153.125
C00662=1089.022,177.119,-70.243,175.836,20.228,153.125
C00663=1089.027,177.368,-70.265,175.839,20.230,153.125
C00664=1089.033,177.616,-70.287,175.842,20.231,153.125
C00665=1089.039,177.866,-70.310,175.844,20.232,153.125
C00666=1089.045,178.115,-70.333,175.847,20.234,153.125
C00667=1089.050,178.363,-70.354,175.850,20.235,153.124
C00668=1089.056,178.612,-70.377,175.852,20.236,153.124
C00669=1089.061,178.862,-70.399,175.855,20.237,153.124
C00670=1089.067,179.111,-70.421,175.858,20.239,153.124
C00671=1089.073,179.359,-70.443,175.860,20.240,153.124
C00672=1089.078,179.609,-70.465,175.863,20.241,153.123
C00673=1089.084,179.857,-70.488,175.865,20.242,153.123
C00674=1089.090,180.107,-70.510,175.868,20.243,153.123
C00675=1089.095,180.355,-70.533,175.870,20.244,153.123
C00676=1089.102,180.604,-70.555,175.873,20.245,153.123
C00677=1089.107,180.853,-70.577,175.876,20.246,153.122
C00678=1089.113,181.102,-70.600,175.878,20.247,153.122
C00679=1089.118,181.352,-70.622,175.881,20.249,153.122
C00680=1089.124,181.599,-70.644,175.884,20.250,153.122
C00681=1089.129,181.849,-70.667,175.886,20.251,153.122
C00682=1089.135,182.098,-70.690,175.889,20.252,153.121
C00683=1089.142,182.346,-70.712,175.892,20.254,153.121
C00684=1089.147,182.596,-70.734,175.895,20.255,153.121
C00685=1089.152,182.844,-70.757,175.897,20.256,153.121
C00686=1089.158,183.093,-70.780,175.901,20.258,153.121
C00687=1089.164,183.342,-70.801,175.904,20.259,153.120
C00688=1089.170,183.591,-70.824,175.906,20.260,153.120
C00689=1089.175,183.840,-70.847,175.909,20.261,153.120
C00690=1089.181,184.090,-70.869,175.912,20.262,153.120
C00691=1089.187,184.338,-70.892,175.914,20.264,153.120
C00692=1089.193,184.586,-70.914,175.917,20.265,153.119
C00693=1089.198,184.836,-70.937,175.920,20.266,153.119
C00694=1089.204,185.085,-70.959,175.922,20.267,153.119
C00695=1089.209,185.334,-70.982,175.925,20.269,153.119
C00696=1089.215,185.583,-71.005,175.928,20.270,153.119
C00697=1089.220,185.831,-71.027,175.930,20.271,153.119
C00698=1089.226,186.080,-71.050,175.933,20.272,153.118
C00699=1089.231,186.329,-71.073,175.936,20.274,153.118
C00700=1089.237,186.578,-71.096,175.938,20.275,153.118
C00701=1089.243,186.827,-71.119,175.941,20.276,153.118
C00702=1089.247,187.076,-71.141,175.944,20.278,153.118
C00703=1089.253,187.325,-71.164,175.946,20.279,153.117
C00704=1089.258,187.574,-71.187,175.949,20.280,153.117
C00705=1089.264,187.823,-71.210,175.952,20.281,153.117
C00706=1089.270,188.072,-71.233,175.954,20.283,153.117
C00707=1089.275,188.320,-71.256,175.957,20.284,153.117
C00708=1089.281,188.569,-71.279,175.960,20.285,153.117
C00709=1089.286,188.818,-71.301,175.962,20.286,153.116
C00710=1089.291,189.067,-71.325,175.965,20.288,153.116
C00711=1089.297,189.316,-71.348,175.968,20.289,153.116
C00712=1089.303,189.565,-71.370,175.970,20.290,153.116
C00713=1089.308,189.813,-71.393,175.974,20.292,153.116
C00714=1089.313,190.062,-71.416,175.977,20.293,153.115
C00715=1089.319,190.311,-71.439,175.979,20.295,153.115
C00716=1089.324,190.560,-71.462,175.982,20.296,153.115
C00717=1089.330,190.809,-71.485,175.984,20.297,153.115
C00718=1089.336,191.058,-71.508,175.987,20.298,153.115
C00719=1089.341,191.307,-71.531,175.990,20.299,153.115
C00720=1089.347,191.584,-71.556,175.993,20.301,153.114
C00721=1089.354,191.861,-71.582,175.996,20.302,153.114
C00722=1089.359,192.138,-71.608,175.999,20.304,153.114
C00723=1089.366,192.415,-71.634,176.002,20.305,153.114
C00724=1089.372,192.664,-71.657,176.005,20.307,153.114
C00725=1089.377,192.912,-71.680,176.008,20.308,153.113
C00726=1089.382,193.161,-71.703,176.011,20.309,153.113
C00727=1089.387,193.410,-71.726,176.013,20.310,153.113
C00728=1089.393,193.659,-71.749,176.016,20.311,153.113
C00729=1089.399,193.908,-71.772,176.018,20.313,153.113
C00730=1089.405,194.157,-71.795,176.021,20.314,153.112
C00731=1089.410,194.406,-71.819,176.024,20.315,153.112
C00732=1089.416,194.654,-71.842,176.027,20.316,153.112
C00733=1089.421,194.903,-71.865,176.029,20.317,153.112
C00734=1089.427,195.152,-71.888,176.033,20.319,153.112
C00735=1089.432,195.401,-71.912,176.036,20.320,153.111
C00736=1089.438,195.650,-71.935,176.038,20.321,153.111
C00737=1089.444,195.899,-71.958,176.041,20.323,153.111
C00738=1089.450,196.148,-71.981,176.044,20.324,153.111
C00739=1089.455,196.397,-72.005,176.046,20.325,153.111
C00740=1089.460,196.646,-72.028,176.049,20.326,153.110
C00741=1089.466,196.894,-72.051,176.052,20.327,153.110
C00742=1089.471,197.143,-72.075,176.054,20.329,153.110
C00743=1089.477,197.392,-72.098,176.058,20.330,153.110
C00744=1089.483,197.641,-72.121,176.061,20.331,153.109
C00745=1089.489,197.889,-72.145,176.063,20.333,153.109
C00746=1089.494,198.138,-72.168,176.066,20.334,153.109
C00747=1089.500,198.387,-72.191,176.069,20.335,153.109
C00748=1089.506,198.636,-72.215,176.072,20.336,153.109
C00749=1089.511,198.885,-72.239,176.074,20.337,153.109
C00750=1089.517,199.134,-72.262,176.077,20.338,153.108
C00751=1089.523,199.383,-72.285,176.080,20.340,153.108
C00752=1089.528,199.632,-72.309,176.083,20.341,153.108
C00753=1089.534,199.880,-72.332,176.086,20.342,153.108
C00754=1089.540,200.129,-72.355,176.089,20.344,153.107
C00755=1089.545,200.378,-72.379,176.092,20.345,153.107
C00756=1089.551,200.627,-72.403,176.094,20.346,153.107
C00757=1089.557,200.875,-72.426,176.097,20.347,153.107
C00758=1089.562,201.125,-72.450,176.100,20.348,153.107
C00759=1089.568,201.374,-72.473,176.102,20.349,153.106
C00760=1089.573,201.622,-72.497,176.106,20.351,153.106
C00761=1089.579,201.871,-72.520,176.109,20.352,153.106
C00762=1089.585,202.119,-72.544,176.111,20.353,153.106
C00763=1089.590,202.369,-72.568,176.114,20.354,153.105
C00764=1089.597,202.618,-72.592,176.117,20.355,153.105
C00765=1089.602,202.867,-72.615,176.120,20.357,153.105
C00766=1089.608,203.115,-72.639,176.123,20.358,153.105
C00767=1089.613,203.364,-72.662,176.126,20.359,153.105
C00768=1089.619,203.613,-72.686,176.129,20.361,153.104
C00769=1089.624,203.862,-72.709,176.131,20.362,153.104
C00770=1089.629,204.110,-72.734,176.134,20.363,153.104
C00771=1089.635,204.359,-72.757,176.137,20.364,153.104
C00772=1089.641,204.609,-72.781,176.140,20.365,153.104
C00773=1089.647,204.857,-72.805,176.143,20.367,153.103
C00774=1089.652,205.106,-72.829,176.146,20.368,153.103
C00775=1089.657,205.355,-72.853,176.149,20.369,153.103
C00776=1089.663,205.603,-72.876,176.151,20.370,153.103
C00777=1089.668,205.852,-72.900,176.154,20.371,153.103
C00778=1089.674,206.100,-72.924,176.157,20.372,153.102
C00779=1089.680,206.350,-72.948,176.160,20.374,153.102
C00780=1089.685,206.599,-72.972,176.163,20.375,153.102
C00781=1089.691,206.847,-72.995,176.166,20.376,153.102
C00782=1089.696,207.096,-73.020,176.168,20.377,153.102
C00783=1089.702,207.344,-73.044,176.171,20.379,153.101
C00784=1089.725,208.367,-73.142,176.241,20.413,153.097
C00785=1089.734,208.748,-73.179,176.245,20.417,153.097
C00786=1089.743,209.129,-73.216,176.249,20.420,153.097
C00787=1089.751,209.511,-73.254,176.254,20.423,153.097
C00788=1089.760,209.892,-73.291,176.257,20.427,153.097
C00789=1089.765,210.141,-73.316,176.260,20.429,153.097
C00790=1089.771,210.390,-73.340,176.263,20.431,153.097
C00791=1089.776,210.639,-73.365,176.266,20.433,153.097
C00792=1089.782,210.887,-73.388,176.269,20.435,153.097
C00793=1089.788,211.136,-73.414,176.271,20.437,153.097
C00794=1089.794,211.384,-73.438,176.274,20.440,153.097
C00795=1089.799,211.633,-73.462,176.277,20.442,153.097
C00796=1089.805,211.882,-73.487,176.280,20.444,153.097
C00797=1089.810,212.131,-73.511,176.282,20.446,153.097
C00798=1089.816,212.379,-73.536,176.284,20.448,153.097
C00799=1089.822,212.628,-73.561,176.288,20.450,153.097
C00800=1089.827,212.877,-73.585,176.290,20.452,153.097
C00801=1089.833,213.126,-73.609,176.293,20.454,153.097
C00802=1089.838,213.375,-73.634,176.296,20.456,153.097
C00803=1089.844,213.623,-73.659,176.299,20.459,153.097
C00804=1089.850,213.872,-73.683,176.301,20.461,153.097
C00805=1089.855,214.121,-73.709,176.305,20.463,153.097
C00806=1089.860,214.369,-73.734,176.307,20.465,153.097
C00807=1089.866,214.618,-73.758,176.310,20.468,153.097
C00808=1089.872,214.867,-73.782,176.312,20.470,153.097
C00809=1089.877,215.115,-73.807,176.316,20.472,153.097
C00810=1089.883,215.364,-73.832,176.318,20.474,153.098
C00811=1089.888,215.613,-73.856,176.321,20.477,153.098
C00812=1089.895,215.862,-73.882,176.324,20.478,153.097
C00813=1089.899,216.111,-73.906,176.327,20.481,153.097
C00814=1089.905,216.360,-73.931,176.329,20.483,153.097
C00815=1089.911,216.608,-73.956,176.332,20.485,153.097
C00816=1089.916,216.856,-73.980,176.335,20.487,153.098
C00817=1089.922,217.105,-74.006,176.338,20.490,153.098
C00818=1089.927,217.354,-74.030,176.340,20.492,153.098
C00819=1089.933,217.603,-74.056,176.344,20.494,153.098
C00820=1089.938,217.851,-74.080,176.346,20.496,153.098
C00821=1089.944,218.100,-74.105,176.349,20.498,153.098
C00822=1089.950,218.349,-74.130,176.351,20.500,153.098
C00823=1089.956,218.597,-74.155,176.355,20.502,153.098
C00824=1089.961,218.847,-74.180,176.357,20.504,153.098
C00825=1089.967,219.095,-74.205,176.360,20.507,153.098
C00826=1089.973,219.344,-74.230,176.363,20.509,153.098
C00827=1089.978,219.592,-74.255,176.366,20.511,153.098
C00828=1089.984,219.841,-74.279,176.368,20.513,153.098
C00829=1089.989,220.090,-74.305,176.371,20.516,153.098
C00830=1089.995,220.339,-74.330,176.374,20.518,153.098
C00831=1090.001,220.588,-74.355,176.377,20.520,153.098
C00832=1090.007,220.836,-74.380,176.380,20.522,153.098
C00833=1090.012,221.085,-74.405,176.383,20.524,153.098
C00834=1090.017,221.333,-74.430,176.385,20.526,153.098
C00835=1090.024,221.582,-74.455,176.388,20.529,153.098
C00836=1090.030,221.831,-74.480,176.391,20.531,153.098
C00837=1090.037,222.216,-74.519,176.396,20.534,153.098
C00838=1090.047,222.601,-74.558,176.399,20.537,153.098
C00839=1090.055,222.986,-74.597,176.404,20.541,153.098
C00840=1090.064,223.371,-74.636,176.408,20.544,153.098
C00841=1090.069,223.620,-74.662,176.411,20.547,153.098
C00842=1090.075,223.868,-74.687,176.414,20.549,153.098
C00843=1090.081,224.117,-74.712,176.417,20.551,153.098
C00844=1090.086,224.366,-74.738,176.419,20.553,153.098
C00845=1090.092,224.614,-74.763,176.422,20.556,153.098
C00846=1090.097,224.863,-74.789,176.425,20.558,153.098
C00847=1090.103,225.111,-74.814,176.428,20.560,153.098
C00848=1090.108,225.360,-74.840,176.430,20.562,153.098
C00849=1090.114,225.610,-74.864,176.434,20.564,153.098
C00850=1090.119,225.858,-74.890,176.436,20.566,153.098
C00851=1090.125,226.107,-74.915,176.439,20.569,153.098
C00852=1090.131,226.356,-74.941,176.443,20.571,153.098
C00853=1090.136,226.603,-74.966,176.445,20.573,153.098
C00854=1090.142,226.852,-74.992,176.448,20.575,153.098
C00855=1090.148,227.101,-75.017,176.450,20.577,153.098
C00856=1090.153,227.349,-75.043,176.454,20.580,153.098
C00857=1090.159,227.598,-75.068,176.456,20.582,153.098
C00858=1090.165,227.847,-75.094,176.459,20.584,153.098
C00859=1090.171,228.096,-75.120,176.461,20.586,153.098
C00860=1090.176,228.344,-75.145,176.465,20.589,153.098
C00861=1090.182,228.593,-75.170,176.468,20.591,153.098
C00862=1090.187,228.842,-75.196,176.470,20.593,153.098
C00863=1090.194,229.090,-75.222,176.474,20.595,153.098
C00864=1090.198,229.339,-75.247,176.476,20.597,153.098
C00865=1090.204,229.588,-75.273,176.479,20.600,153.098
C00866=1090.210,229.836,-75.299,176.482,20.602,153.098
C00867=1090.216,230.085,-75.325,176.485,20.604,153.098
C00868=1090.221,230.333,-75.349,176.488,20.607,153.098
C00869=1090.227,230.582,-75.375,176.490,20.609,153.098
C00870=1090.232,230.831,-75.401,176.494,20.611,153.098
C00871=1090.239,231.079,-75.427,176.496,20.613,153.098
C00872=1090.244,231.327,-75.453,176.499,20.615,153.098
C00873=1090.249,231.576,-75.479,176.502,20.618,153.098
C00874=1090.255,231.825,-75.504,176.505,20.620,153.098
C00875=1090.261,232.074,-75.530,176.508,20.622,153.098
C00876=1090.266,232.323,-75.556,176.510,20.624,153.098
C00877=1090.271,232.571,-75.582,176.513,20.627,153.098
C00878=1090.278,232.819,-75.608,176.516,20.629,153.098
C00879=1090.283,233.068,-75.634,176.519,20.631,153.098
C00880=1090.288,233.317,-75.660,176.522,20.634,153.099
C00881=1090.294,233.566,-75.686,176.525,20.636,153.099
C00882=1090.300,233.814,-75.711,176.528,20.638,153.099
C00883=1090.305,234.063,-75.737,176.530,20.640,153.099
C00884=1090.311,234.311,-75.764,176.533,20.643,153.099
C00885=1090.317,234.560,-75.790,176.536,20.645,153.099
C00886=1090.322,234.809,-75.816,176.539,20.647,153.099
C00887=1090.328,235.057,-75.842,176.542,20.649,153.099
C00888=1090.333,235.305,-75.867,176.544,20.651,153.099
C00889=1090.341,235.683,-75.907,176.549,20.655,153.099
C00890=1090.350,236.059,-75.947,176.553,20.658,153.099
C00891=1090.359,236.435,-75.986,176.558,20.662,153.099
C00892=1090.367,236.812,-76.026,176.562,20.665,153.099
C00893=1090.372,237.060,-76.052,176.565,20.668,153.099
C00894=1090.378,237.309,-76.078,176.568,20.670,153.099
C00895=1090.384,237.557,-76.104,176.571,20.672,153.099
C00896=1090.390,237.806,-76.130,176.574,20.675,153.099
C00897=1090.396,238.054,-76.156,176.577,20.677,153.099
C00898=1090.401,238.303,-76.182,176.579,20.679,153.099
C00899=1090.407,238.552,-76.209,176.583,20.681,153.099
C00900=1090.412,238.801,-76.235,176.585,20.683,153.099
C00901=1090.418,239.049,-76.262,176.588,20.686,153.099
C00902=1090.424,239.298,-76.288,176.591,20.688,153.099
C00903=1090.429,239.546,-76.314,176.594,20.690,153.099
C00904=1090.435,239.795,-76.341,176.597,20.693,153.099
C00905=1090.441,240.044,-76.367,176.600,20.695,153.099
C00906=1090.446,240.291,-76.393,176.603,20.697,153.099
C00907=1090.452,240.540,-76.420,176.606,20.700,153.099
C00908=1090.457,240.789,-76.446,176.609,20.702,153.099
C00909=1090.463,241.037,-76.472,176.611,20.704,153.099
C00910=1090.468,241.286,-76.498,176.614,20.707,153.099
C00911=1090.474,241.534,-76.525,176.617,20.709,153.099
C00912=1090.480,241.783,-76.551,176.620,20.711,153.099
C00913=1090.486,242.031,-76.578,176.623,20.713,153.099
C00914=1090.491,242.280,-76.604,176.626,20.715,153.099
C00915=1090.497,242.529,-76.631,176.629,20.718,153.099
C00916=1090.503,242.777,-76.657,176.632,20.720,153.099
C00917=1090.508,243.025,-76.684,176.634,20.722,153.100
C00918=1090.514,243.274,-76.710,176.638,20.725,153.100
C00919=1090.519,243.523,-76.737,176.641,20.727,153.100
C00920=1090.525,243.771,-76.764,176.643,20.729,153.100
C00921=1090.530,244.020,-76.790,176.646,20.732,153.100
C00922=1090.536,244.268,-76.817,176.650,20.734,153.100
C00923=1090.542,244.517,-76.843,176.652,20.737,153.100
C00924=1090.547,244.765,-76.870,176.655,20.739,153.100
C00925=1090.553,245.015,-76.897,176.658,20.741,153.100
C00926=1090.559,245.263,-76.924,176.660,20.743,153.100
C00927=1090.565,245.511,-76.951,176.664,20.746,153.100
C00928=1090.570,245.760,-76.977,176.667,20.748,153.100
C00929=1090.575,246.008,-77.005,176.669,20.750,153.100
C00930=1090.581,246.257,-77.031,176.672,20.753,153.100
C00931=1090.587,246.505,-77.058,176.676,20.755,153.100
C00932=1090.592,246.754,-77.084,176.678,20.757,153.100
C00933=1090.597,247.003,-77.111,176.681,20.760,153.100
C00934=1090.603,247.251,-77.138,176.684,20.762,153.100
C00935=1090.609,247.500,-77.164,176.687,20.765,153.100
C00936=1090.614,247.748,-77.192,176.690,20.767,153.100
C00937=1090.620,247.997,-77.218,176.693,20.769,153.100
C00938=1090.626,248.245,-77.245,176.696,20.772,153.100
C00939=1090.631,248.493,-77.273,176.699,20.774,153.100
C00940=1090.637,248.741,-77.299,176.702,20.777,153.101
C00941=1090.645,249.112,-77.340,176.706,20.780,153.101
C00942=1090.653,249.481,-77.379,176.710,20.784,153.101
C00943=1090.662,249.851,-77.420,176.715,20.788,153.101
C00944=1090.670,250.220,-77.460,176.719,20.791,153.101
C00945=1090.675,250.469,-77.487,176.722,20.794,153.101
C00946=1090.681,250.718,-77.514,176.725,20.796,153.101
C00947=1090.686,250.966,-77.542,176.728,20.798,153.101
C00948=1090.692,251.214,-77.569,176.731,20.800,153.101
C00949=1090.697,251.463,-77.596,176.734,20.803,153.101
C00950=1090.703,251.711,-77.623,176.736,20.805,153.101
C00951=1090.708,251.960,-77.650,176.739,20.808,153.101
C00952=1090.714,252.208,-77.677,176.743,20.810,153.101
C00953=1090.720,252.457,-77.705,176.746,20.813,153.101
C00954=1090.725,252.705,-77.731,176.748,20.815,153.101
C00955=1090.731,252.954,-77.759,176.751,20.818,153.101
C00956=1090.737,253.202,-77.786,176.754,20.820,153.102
C00957=1090.742,253.450,-77.813,176.757,20.822,153.102
C00958=1090.748,253.700,-77.840,176.760,20.824,153.102
C00959=1090.753,253.948,-77.868,176.763,20.827,153.102
C00960=1090.759,254.196,-77.895,176.766,20.829,153.102
C00961=1090.764,254.445,-77.922,176.769,20.832,153.102
C00962=1090.770,254.692,-77.950,176.772,20.834,153.102
C00963=1090.776,254.942,-77.977,176.775,20.837,153.102
C00964=1090.782,255.189,-78.005,176.778,20.839,153.102
C00965=1090.787,255.438,-78.032,176.781,20.841,153.102
C00966=1090.792,255.686,-78.060,176.784,20.844,153.102
C00967=1090.799,255.935,-78.087,176.787,20.847,153.102
C00968=1090.804,256.184,-78.114,176.790,20.849,153.102
C00969=1090.810,256.432,-78.141,176.792,20.851,153.102
C00970=1090.815,256.680,-78.169,176.796,20.853,153.102
C00971=1090.821,256.929,-78.197,176.799,20.856,153.102
C00972=1090.827,257.177,-78.224,176.802,20.858,153.102
C00973=1090.832,257.425,-78.252,176.804,20.861,153.102
C00974=1090.839,257.674,-78.279,176.807,20.863,153.102
C00975=1090.844,257.923,-78.306,176.811,20.866,153.102
C00976=1090.849,258.171,-78.334,176.814,20.868,153.103
C00977=1090.855,258.420,-78.361,176.816,20.870,153.103
C00978=1090.861,258.668,-78.389,176.819,20.873,153.103
C00979=1090.867,258.915,-78.417,176.822,20.875,153.103
C00980=1090.872,259.165,-78.444,176.826,20.878,153.103
C00981=1090.878,259.413,-78.472,176.828,20.880,153.103
C00982=1090.884,259.661,-78.499,176.831,20.882,153.103
C00983=1090.889,259.910,-78.527,176.834,20.885,153.103
C00984=1090.895,260.158,-78.555,176.838,20.887,153.103
C00985=1090.901,260.407,-78.582,176.840,20.889,153.103
C00986=1090.907,260.655,-78.610,176.843,20.892,153.103
C00987=1090.912,260.903,-78.638,176.846,20.895,153.103
C00988=1090.919,261.152,-78.666,176.849,20.897,153.103
C00989=1090.924,261.400,-78.693,176.853,20.899,153.103
C00990=1090.930,261.649,-78.722,176.855,20.901,153.103
C00991=1090.935,261.897,-78.749,176.858,20.904,153.103
C00992=1090.941,262.145,-78.777,176.861,20.907,153.103
C00993=1090.950,262.512,-78.818,176.866,20.910,153.103
C00994=1090.958,262.879,-78.859,176.870,20.914,153.104
C00995=1090.967,263.245,-78.901,176.875,20.918,153.104
C00996=1090.975,263.612,-78.942,176.879,20.921,153.104
C00997=1090.981,263.861,-78.969,176.882,20.923,153.104
C00998=1090.987,264.109,-78.997,176.885,20.926,153.104
C00999=1090.993,264.358,-79.025,176.888,20.928,153.104
C01000=1090.998,264.606,-79.053,176.891,20.930,153.104
C01001=1091.003,264.854,-79.081,176.894,20.933,153.104
C01002=1091.009,265.103,-79.109,176.897,20.936,153.104
C01003=1091.015,265.351,-79.137,176.900,20.938,153.104
C01004=1091.021,265.599,-79.166,176.903,20.941,153.104
C01005=1091.026,265.847,-79.193,176.905,20.943,153.104
C01006=1091.032,266.096,-79.222,176.909,20.945,153.104
C01007=1091.037,266.344,-79.250,176.912,20.948,153.104
C01008=1091.043,266.593,-79.278,176.915,20.951,153.105
C01009=1091.049,266.841,-79.306,176.918,20.953,153.105
C01010=1091.055,267.090,-79.334,176.921,20.956,153.105
C01011=1091.060,267.338,-79.362,176.923,20.958,153.105
C01012=1091.065,267.586,-79.390,176.927,20.961,153.105
C01013=1091.071,267.835,-79.419,176.930,20.963,153.105
C01014=1091.077,268.082,-79.447,176.933,20.966,153.105
C01015=1091.083,268.331,-79.476,176.936,20.968,153.105
C01016=1091.089,268.580,-79.504,176.939,20.971,153.105
C01017=1091.094,268.828,-79.532,176.941,20.973,153.105
C01018=1091.100,269.076,-79.560,176.945,20.976,153.105
C01019=1091.105,269.324,-79.588,176.948,20.978,153.105
C01020=1091.112,269.573,-79.617,176.951,20.981,153.105
C01021=1091.117,269.821,-79.645,176.954,20.984,153.106
C01022=1091.123,270.069,-79.674,176.957,20.986,153.106
C01023=1091.127,270.318,-79.702,176.960,20.988,153.106
C01024=1091.134,270.566,-79.731,176.963,20.991,153.106
C01025=1091.139,270.814,-79.759,176.966,20.994,153.106
C01026=1091.145,271.063,-79.787,176.969,20.996,153.106
C01027=1091.150,271.311,-79.815,176.972,20.999,153.106
C01028=1091.157,271.559,-79.844,176.975,21.002,153.106
C01029=1091.162,271.808,-79.873,176.978,21.004,153.106
C01030=1091.167,272.056,-79.901,176.981,21.007,153.106
C01031=1091.173,272.304,-79.930,176.984,21.009,153.106
C01032=1091.179,272.552,-79.958,176.987,21.011,153.106
C01033=1091.185,272.800,-79.987,176.990,21.014,153.107
C01034=1091.190,273.049,-80.016,176.993,21.017,153.107
C01035=1091.196,273.297,-80.044,176.996,21.020,153.107
C01036=1091.202,273.545,-80.073,176.999,21.022,153.107
C01037=1091.207,273.794,-80.101,177.002,21.024,153.107
C01038=1091.213,274.042,-80.130,177.005,21.027,153.107
C01039=1091.219,274.291,-80.159,177.008,21.029,153.107
C01040=1091.224,274.538,-80.188,177.011,21.032,153.107
C01041=1091.230,274.787,-80.216,177.014,21.035,153.107
C01042=1091.235,275.035,-80.245,177.017,21.038,153.107
C01043=1091.241,275.283,-80.274,177.020,21.040,153.108
C01044=1091.247,275.532,-80.303,177.023,21.043,153.108
C01045=1091.255,275.901,-80.345,177.027,21.047,153.108
C01046=1091.264,276.270,-80.389,177.032,21.050,153.108
C01047=1091.272,276.640,-80.431,177.037,21.054,153.108
C01048=1091.281,277.009,-80.475,177.041,21.058,153.108
C01049=1091.285,277.258,-80.503,177.044,21.061,153.108
C01050=1091.292,277.506,-80.532,177.047,21.064,153.109
C01051=1091.298,277.755,-80.561,177.050,21.066,153.109
C01052=1091.303,278.003,-80.590,177.053,21.069,153.109
C01053=1091.309,278.250,-80.619,177.056,21.071,153.109
C01054=1091.314,278.499,-80.649,177.059,21.074,153.109
C01055=1091.320,278.748,-80.677,177.062,21.077,153.109
C01056=1091.325,278.995,-80.706,177.065,21.080,153.109
C01057=1091.331,279.244,-80.735,177.068,21.082,153.109
C01058=1091.338,279.492,-80.764,177.071,21.085,153.109
C01059=1091.343,279.741,-80.793,177.074,21.087,153.110
C01060=1091.349,279.988,-80.822,177.077,21.090,153.110
C01061=1091.354,280.237,-80.851,177.080,21.093,153.110
C01062=1091.360,280.485,-80.880,177.083,21.095,153.110
C01063=1091.366,280.733,-80.910,177.086,21.098,153.110
C01064=1091.371,280.981,-80.938,177.090,21.101,153.110
C01065=1091.377,281.230,-80.968,177.093,21.104,153.110
C01066=1091.383,281.478,-80.997,177.096,21.106,153.110
C01067=1091.388,281.726,-81.026,177.099,21.109,153.110
C01068=1091.393,281.974,-81.056,177.102,21.112,153.111
C01069=1091.400,282.222,-81.085,177.104,21.114,153.111
C01070=1091.405,282.471,-81.114,177.107,21.117,153.111
C01071=1091.411,282.719,-81.144,177.110,21.120,153.111
C01072=1091.416,282.966,-81.173,177.113,21.122,153.111
C01073=1091.422,283.215,-81.202,177.117,21.125,153.111
C01074=1091.427,283.463,-81.232,177.120,21.128,153.111
C01075=1091.434,283.711,-81.261,177.123,21.131,153.111
C01076=1091.439,283.960,-81.291,177.126,21.133,153.112
C01077=1091.444,284.208,-81.320,177.129,21.136,153.112
C01078=1091.450,284.456,-81.349,177.132,21.139,153.112
C01079=1091.456,284.704,-81.379,177.135,21.141,153.112
C01080=1091.461,284.953,-81.408,177.138,21.144,153.112
C01081=1091.467,285.201,-81.437,177.141,21.147,153.112
C01082=1091.472,285.448,-81.466,177.144,21.150,153.112
C01083=1091.478,285.697,-81.496,177.147,21.153,153.112
C01084=1091.484,285.945,-81.525,177.149,21.155,153.113
C01085=1091.490,286.193,-81.555,177.153,21.158,153.113
C01086=1091.495,286.441,-81.585,177.156,21.160,153.113
C01087=1091.501,286.690,-81.615,177.159,21.163,153.113
C01088=1091.507,286.938,-81.644,177.162,21.166,153.113
C01089=1091.512,287.186,-81.673,177.165,21.169,153.113
C01090=1091.518,287.433,-81.703,177.168,21.172,153.113
C01091=1091.523,287.682,-81.733,177.171,21.174,153.114
C01092=1091.530,287.930,-81.762,177.174,21.177,153.114
C01093=1091.535,288.178,-81.792,177.177,21.180,153.114
C01094=1091.541,288.426,-81.822,177.180,21.183,153.114
C01095=1091.547,288.675,-81.852,177.183,21.186,153.114
C01096=1091.553,288.923,-81.881,177.187,21.188,153.114
C01097=1091.561,289.301,-81.927,177.191,21.192,153.114
C01098=1091.570,289.681,-81.972,177.196,21.197,153.115
C01099=1091.579,290.059,-82.018,177.200,21.201,153.115
C01100=1091.588,290.438,-82.063,177.205,21.205,153.115
C01101=1091.593,290.687,-82.092,177.208,21.208,153.115
C01102=1091.599,290.934,-82.123,177.211,21.211,153.115
C01103=1091.604,291.183,-82.152,177.214,21.214,153.116
C01104=1091.610,291.431,-82.183,177.217,21.217,153.116
C01105=1091.616,291.679,-82.212,177.220,21.219,153.116
C01106=1091.621,291.927,-82.243,177.223,21.222,153.116
C01107=1091.627,292.175,-82.272,177.226,21.225,153.116
C01108=1091.633,292.423,-82.303,177.229,21.228,153.116
C01109=1091.638,292.672,-82.332,177.232,21.231,153.117
C01110=1091.644,292.919,-82.363,177.235,21.234,153.117
C01111=1091.650,293.168,-82.392,177.238,21.237,153.117
C01112=1091.655,293.416,-82.423,177.241,21.239,153.117
C01113=1091.661,293.664,-82.453,177.244,21.242,153.117
C01114=1091.667,293.912,-82.483,177.248,21.245,153.117
C01115=1091.673,294.160,-82.513,177.251,21.248,153.117
C01116=1091.678,294.408,-82.543,177.254,21.251,153.118
C01117=1091.684,294.656,-82.573,177.257,21.253,153.118
C01118=1091.690,294.904,-82.603,177.260,21.256,153.118
C01119=1091.695,295.152,-82.633,177.263,21.259,153.118
C01120=1091.701,295.400,-82.663,177.266,21.262,153.118
C01121=1091.707,295.648,-82.694,177.269,21.265,153.119
C01122=1091.712,295.896,-82.723,177.272,21.268,153.119
C01123=1091.718,296.145,-82.754,177.275,21.271,153.119
C01124=1091.723,296.392,-82.785,177.279,21.274,153.119
C01125=1091.729,296.640,-82.815,177.282,21.277,153.119
C01126=1091.735,296.888,-82.845,177.285,21.280,153.119
C01127=1091.741,297.137,-82.875,177.288,21.283,153.120
C01128=1091.747,297.385,-82.906,177.291,21.286,153.120
C01129=1091.753,297.633,-82.936,177.294,21.289,153.120
C01130=1091.758,297.881,-82.967,177.297,21.292,153.120
C01131=1091.764,298.129,-82.997,177.300,21.295,153.120
C01132=1091.769,298.377,-83.027,177.303,21.297,153.120
C01133=1091.775,298.625,-83.057,177.306,21.300,153.121
C01134=1091.780,298.873,-83.088,177.309,21.303,153.121
C01135=1091.786,299.121,-83.119,177.312,21.307,153.121
C01136=1091.791,299.369,-83.149,177.315,21.310,153.121
C01137=1091.797,299.617,-83.180,177.318,21.312,153.122
C01138=1091.803,299.865,-83.210,177.321,21.315,153.122
C01139=1091.808,300.113,-83.241,177.324,21.318,153.122
C01140=1091.814,300.361,-83.272,177.327,21.322,153.122
C01141=1091.820,300.609,-83.302,177.330,21.324,153.122
C01142=1091.825,300.857,-83.333,177.334,21.328,153.123
C01143=1091.831,301.105,-83.363,177.337,21.331,153.123
C01144=1091.836,301.353,-83.394,177.340,21.334,153.123
C01145=1091.842,301.601,-83.425,177.343,21.337,153.123
C01146=1091.847,301.849,-83.456,177.346,21.340,153.123
C01147=1091.853,302.097,-83.486,177.349,21.343,153.124
C01148=1091.859,302.346,-83.517,177.351,21.346,153.124
C01149=1091.867,302.738,-83.565,177.357,21.351,153.124
C01150=1091.876,303.131,-83.614,177.361,21.356,153.125
C01151=1091.885,303.524,-83.664,177.366,21.360,153.125
C01152=1091.894,303.917,-83.712,177.371,21.365,153.125
C01153=1091.900,304.165,-83.743,177.374,21.368,153.125
C01154=1091.905,304.412,-83.773,177.377,21.371,153.126
C01155=1091.911,304.661,-83.805,177.380,21.375,153.126
C01156=1091.917,304.909,-83.836,177.383,21.377,153.126
C01157=1091.922,305.157,-83.867,177.387,21.381,153.126
C01158=1091.928,305.404,-83.897,177.390,21.384,153.127
C01159=1091.934,305.653,-83.929,177.393,21.387,153.127
C01160=1091.940,305.900,-83.960,177.396,21.390,153.127
C01161=1091.945,306.149,-83.990,177.399,21.393,153.127
C01162=1091.951,306.396,-84.022,177.402,21.396,153.127
C01163=1091.957,306.645,-84.053,177.405,21.399,153.128
C01164=1091.963,306.892,-84.083,177.407,21.403,153.128
C01165=1091.968,307.140,-84.115,177.411,21.406,153.128
C01166=1091.973,307.388,-84.146,177.414,21.409,153.128
C01167=1091.979,307.637,-84.177,177.417,21.412,153.129
C01168=1091.985,307.884,-84.208,177.420,21.415,153.129
C01169=1091.991,308.132,-84.239,177.423,21.418,153.129
C01170=1091.997,308.380,-84.271,177.426,21.421,153.129
C01171=1092.002,308.628,-84.301,177.429,21.424,153.129
C01172=1092.008,308.876,-84.333,177.432,21.427,153.130
C01173=1092.014,309.124,-84.364,177.436,21.431,153.130
C01174=1092.020,309.372,-84.395,177.439,21.434,153.130
C01175=1092.025,309.620,-84.426,177.442,21.437,153.130
C01176=1092.031,309.868,-84.457,177.445,21.440,153.131
C01177=1092.037,310.116,-84.488,177.448,21.443,153.131
C01178=1092.043,310.364,-84.520,177.451,21.446,153.131
C01179=1092.049,310.611,-84.551,177.454,21.449,153.131
C01180=1092.054,310.860,-84.583,177.457,21.453,153.132
C01181=1092.060,311.107,-84.614,177.460,21.456,153.132
C01182=1092.066,311.355,-84.645,177.463,21.459,153.132
C01183=1092.072,311.604,-84.677,177.466,21.462,153.132
C01184=1092.077,311.851,-84.708,177.469,21.465,153.133
C01185=1092.083,312.100,-84.739,177.472,21.468,153.133
C01186=1092.089,312.347,-84.771,177.476,21.472,153.133
C01187=1092.095,312.595,-84.803,177.479,21.475,153.133
C01188=1092.101,312.842,-84.834,177.482,21.478,153.133
C01189=1092.106,313.091,-84.865,177.485,21.481,153.134
C01190=1092.112,313.339,-84.897,177.488,21.484,153.134
C01191=1092.119,313.587,-84.928,177.491,21.487,153.134
C01192=1092.124,313.834,-84.960,177.495,21.491,153.134
C01193=1092.130,314.083,-84.991,177.498,21.494,153.135
C01194=1092.136,314.330,-85.022,177.500,21.497,153.135
C01195=1092.142,314.579,-85.054,177.503,21.500,153.135
C01196=1092.147,314.826,-85.086,177.506,21.503,153.136
C01197=1092.153,315.074,-85.118,177.509,21.506,153.136
C01198=1092.159,315.322,-85.150,177.513,21.510,153.136
C01199=1092.164,315.571,-85.181,177.516,21.513,153.136
C01200=1092.170,315.818,-85.213,177.519,21.517,153.137
C01201=1092.179,316.214,-85.263,177.524,21.522,153.137
C01202=1092.188,316.609,-85.314,177.528,21.527,153.138
C01203=1092.197,317.005,-85.365,177.533,21.533,153.138
C01204=1092.205,317.400,-85.416,177.538,21.538,153.139
C01205=1092.211,317.648,-85.448,177.541,21.542,153.139
C01206=1092.217,317.896,-85.480,177.544,21.545,153.139
C01207=1092.223,318.144,-85.512,177.547,21.548,153.140
C01208=1092.228,318.391,-85.544,177.551,21.552,153.140
C01209=1092.234,318.640,-85.576,177.553,21.556,153.140
C01210=1092.239,318.888,-85.608,177.556,21.558,153.140
C01211=1092.245,319.136,-85.640,177.559,21.562,153.141
C01212=1092.251,319.384,-85.672,177.562,21.565,153.141
C01213=1092.256,319.631,-85.703,177.566,21.569,153.141
C01214=1092.262,319.879,-85.736,177.569,21.572,153.142
C01215=1092.268,320.126,-85.768,177.572,21.576,153.142
C01216=1092.273,320.375,-85.801,177.574,21.579,153.142
C01217=1092.279,320.623,-85.833,177.578,21.583,153.143
C01218=1092.284,320.871,-85.864,177.581,21.586,153.143
C01219=1092.290,321.119,-85.896,177.584,21.589,153.143
C01220=1092.296,321.366,-85.929,177.587,21.593,153.144
C01221=1092.302,321.614,-85.961,177.590,21.597,153.144
C01222=1092.307,321.863,-85.993,177.593,21.600,153.144
C01223=1092.313,322.110,-86.025,177.596,21.603,153.145
C01224=1092.319,322.358,-86.058,177.599,21.607,153.145
C01225=1092.325,322.606,-86.090,177.603,21.610,153.145
C01226=1092.330,322.854,-86.122,177.605,21.614,153.145
C01227=1092.336,323.101,-86.155,177.608,21.617,153.146
C01228=1092.342,323.350,-86.187,177.611,21.620,153.146
C01229=1092.347,323.597,-86.218,177.615,21.624,153.146
C01230=1092.353,323.845,-86.252,177.618,21.628,153.147
C01231=1092.359,324.093,-86.284,177.621,21.631,153.147
C01232=1092.365,324.340,-86.316,177.623,21.634,153.147
C01233=1092.371,324.588,-86.348,177.627,21.639,153.148
C01234=1092.376,324.837,-86.381,177.630,21.642,153.148
C01235=1092.382,325.084,-86.414,177.633,21.645,153.149
C01236=1092.388,325.332,-86.445,177.636,21.649,153.149
C01237=1092.394,325.580,-86.478,177.639,21.652,153.149
C01238=1092.399,325.828,-86.511,177.642,21.656,153.149
C01239=1092.405,326.076,-86.543,177.645,21.659,153.150
C01240=1092.411,326.323,-86.575,177.649,21.663,153.150
C01241=1092.416,326.571,-86.608,177.651,21.666,153.150
C01242=1092.422,326.819,-86.640,177.654,21.670,153.151
C01243=1092.429,327.067,-86.673,177.658,21.674,153.151
C01244=1092.434,327.315,-86.706,177.661,21.677,153.152
C01245=1092.440,327.562,-86.738,177.664,21.681,153.152
C01246=1092.446,327.810,-86.771,177.666,21.684,153.152
C01247=1092.451,328.058,-86.804,177.670,21.688,153.153
C01248=1092.457,328.306,-86.836,177.673,21.691,153.153
C01249=1092.464,328.554,-86.869,177.676,21.695,153.153
C01250=1092.469,328.801,-86.902,177.679,21.699,153.154
C01251=1092.475,329.050,-86.934,177.682,21.702,153.154
C01252=1092.480,329.297,-86.967,177.685,21.706,153.154
C01253=1092.490,329.685,-87.019,177.690,21.711,153.155
C01254=1092.498,330.075,-87.070,177.695,21.717,153.155
C01255=1092.508,330.463,-87.121,177.700,21.723,153.156
C01256=1092.517,330.852,-87.173,177.705,21.729,153.157
C01257=1092.523,331.099,-87.206,177.708,21.732,153.157
C01258=1092.529,331.347,-87.239,177.711,21.736,153.157
C01259=1092.535,331.595,-87.271,177.714,21.739,153.158
C01260=1092.541,331.843,-87.304,177.717,21.743,153.158
C01261=1092.547,332.091,-87.337,177.720,21.747,153.158
C01262=1092.552,332.339,-87.370,177.723,21.751,153.159
C01263=1092.558,332.586,-87.403,177.726,21.754,153.159
C01264=1092.564,332.834,-87.437,177.729,21.758,153.160
C01265=1092.570,333.082,-87.470,177.733,21.762,153.160
C01266=1092.575,333.329,-87.502,177.735,21.766,153.161
C01267=1092.581,333.577,-87.536,177.738,21.769,153.161
C01268=1092.586,333.825,-87.569,177.742,21.773,153.161
C01269=1092.593,334.072,-87.602,177.744,21.777,153.162
C01270=1092.598,334.320,-87.635,177.748,21.781,153.162
C01271=1092.604,334.568,-87.668,177.751,21.784,153.163
C01272=1092.609,334.816,-87.702,177.753,21.788,153.163
C01273=1092.616,335.064,-87.734,177.757,21.792,153.163
C01274=1092.621,335.312,-87.768,177.760,21.796,153.164
C01275=1092.627,335.559,-87.801,177.763,21.800,153.164
C01276=1092.633,335.806,-87.835,177.766,21.804,153.165
C01277=1092.639,336.054,-87.868,177.769,21.807,153.165
C01278=1092.644,336.302,-87.901,177.772,21.811,153.165
C01279=1092.650,336.550,-87.935,177.775,21.815,153.166
C01280=1092.656,336.798,-87.968,177.779,21.820,153.166
C01281=1092.662,337.046,-88.001,177.781,21.823,153.167
C01282=1092.668,337.293,-88.035,177.784,21.827,153.167
C01283=1092.673,337.541,-88.068,177.788,21.831,153.168
C01284=1092.679,337.789,-88.101,177.790,21.835,153.168
C01285=1092.685,338.036,-88.134,177.794,21.838,153.168
C01286=1092.691,338.284,-88.168,177.797,21.842,153.169
C01287=1092.697,338.531,-88.202,177.800,21.846,153.169
C01288=1092.702,338.779,-88.235,177.803,21.850,153.170
C01289=1092.708,339.027,-88.269,177.806,21.854,153.170
C01290=1092.714,339.275,-88.302,177.809,21.858,153.171
C01291=1092.719,339.522,-88.336,177.812,21.862,153.171
C01292=1092.725,339.770,-88.370,177.815,21.866,153.172
C01293=1092.730,340.018,-88.403,177.818,21.870,153.172
C01294=1092.736,340.265,-88.437,177.821,21.874,153.173
C01295=1092.743,340.514,-88.471,177.824,21.878,153.173
C01296=1092.748,340.761,-88.504,177.828,21.882,153.174
C01297=1092.754,341.009,-88.538,177.830,21.886,153.174
C01298=1092.759,341.257,-88.571,177.834,21.890,153.174
C01299=1092.765,341.504,-88.606,177.837,21.894,153.175
C01300=1092.771,341.752,-88.639,177.840,21.899,153.176
C01301=1092.777,341.999,-88.673,177.843,21.903,153.176
C01302=1092.782,342.247,-88.706,177.845,21.906,153.176
C01303=1092.788,342.494,-88.740,177.849,21.911,153.177
C01304=1092.795,342.742,-88.775,177.851,21.914,153.177
C01305=1092.803,343.124,-88.826,177.856,21.921,153.178
C01306=1092.812,343.507,-88.879,177.861,21.927,153.179
C01307=1092.821,343.890,-88.931,177.866,21.934,153.180
C01308=1092.830,344.273,-88.983,177.871,21.940,153.180
C01309=1092.837,344.521,-89.018,177.874,21.944,153.181
C01310=1092.842,344.768,-89.051,177.877,21.948,153.181
C01311=1092.847,345.016,-89.086,177.880,21.953,153.182
C01312=1092.853,345.263,-89.120,177.883,21.956,153.182
C01313=1092.859,345.511,-89.154,177.886,21.961,153.183
C01314=1092.865,345.759,-89.188,177.889,21.965,153.183
C01315=1092.871,346.007,-89.222,177.892,21.969,153.184
C01316=1092.876,346.254,-89.256,177.895,21.973,153.185
C01317=1092.882,346.501,-89.290,177.899,21.978,153.185
C01318=1092.888,346.749,-89.324,177.901,21.982,153.186
C01319=1092.894,346.997,-89.359,177.905,21.986,153.186
C01320=1092.899,347.245,-89.393,177.908,21.991,153.187
C01321=1092.905,347.492,-89.427,177.911,21.994,153.187
C01322=1092.911,347.739,-89.461,177.914,21.999,153.188
C01323=1092.917,347.987,-89.495,177.917,22.003,153.188
C01324=1092.923,348.235,-89.530,177.920,22.008,153.189
C01325=1092.928,348.482,-89.564,177.922,22.012,153.189
C01326=1092.934,348.730,-89.598,177.926,22.016,153.190
C01327=1092.940,348.978,-89.633,177.929,22.020,153.190
C01328=1092.946,349.225,-89.667,177.932,22.025,153.191
C01329=1092.952,349.472,-89.701,177.935,22.029,153.191
C01330=1092.957,349.720,-89.736,177.938,22.033,153.192
C01331=1092.963,349.968,-89.770,177.941,22.038,153.193
C01332=1092.969,350.215,-89.804,177.944,22.042,153.193
C01333=1092.974,350.463,-89.839,177.947,22.047,153.194
C01334=1092.981,350.710,-89.874,177.950,22.051,153.194
C01335=1092.986,350.958,-89.909,177.953,22.055,153.195
C01336=1092.992,351.205,-89.943,177.957,22.060,153.195
C01337=1092.998,351.453,-89.977,177.959,22.064,153.196
C01338=1093.004,351.701,-90.012,177.963,22.069,153.197
C01339=1093.009,351.948,-90.046,177.965,22.073,153.197
C01340=1093.015,352.196,-90.082,177.968,22.077,153.198
C01341=1093.021,352.443,-90.116,177.972,22.082,153.198
C01342=1093.027,352.690,-90.150,177.975,22.086,153.199
C01343=1093.033,352.939,-90.185,177.978,22.091,153.199
C01344=1093.039,353.185,-90.220,177.980,22.095,153.200
C01345=1093.045,353.434,-90.255,177.984,22.099,153.201
C01346=1093.051,353.681,-90.289,177.987,22.104,153.201
C01347=1093.056,353.928,-90.324,177.990,22.108,153.202
C01348=1093.062,354.176,-90.359,177.993,22.113,153.202
C01349=1093.068,354.423,-90.393,177.996,22.118,153.203
C01350=1093.073,354.670,-90.428,177.999,22.122,153.204
C01351=1093.080,354.918,-90.463,178.002,22.127,153.204
C01352=1093.085,355.165,-90.498,178.005,22.131,153.205
C01353=1093.091,355.414,-90.533,178.008,22.136,153.206
C01354=1093.097,355.661,-90.567,178.011,22.141,153.206
C01355=1093.102,355.908,-90.603,178.014,22.145,153.207
C01356=1093.108,356.156,-90.637,178.017,22.149,153.207
C01357=1093.117,356.541,-90.692,178.022,22.157,153.209
C01358=1093.126,356.926,-90.746,178.027,22.164,153.209
C01359=1093.135,357.312,-90.801,178.032,22.171,153.210
C01360=1093.144,357.696,-90.856,178.036,22.178,153.211
C01361=1093.150,357.944,-90.891,178.039,22.184,153.212
C01362=1093.156,358.191,-90.926,178.042,22.188,153.213
C01363=1093.162,358.439,-90.961,178.045,22.192,153.213
C01364=1093.167,358.686,-90.996,178.048,22.197,153.214
C01365=1093.174,358.934,-91.031,178.052,22.202,153.215
C01366=1093.179,359.181,-91.066,178.054,22.207,153.215
C01367=1093.185,359.429,-91.101,178.057,22.211,153.216
C01368=1093.191,359.676,-91.137,178.061,22.216,153.217
C01369=1093.197,359.923,-91.172,178.063,22.221,153.217
C01370=1093.203,360.171,-91.207,178.067,22.225,153.218
C01371=1093.209,360.419,-91.242,178.070,22.231,153.219
C01372=1093.214,360.666,-91.278,178.072,22.235,153.219
C01373=1093.220,360.913,-91.313,178.075,22.240,153.220
C01374=1093.226,361.160,-91.348,178.079,22.245,153.221
C01375=1093.232,361.408,-91.384,178.082,22.250,153.222
C01376=1093.238,361.656,-91.419,178.084,22.254,153.222
C01377=1093.243,361.903,-91.454,178.088,22.259,153.223
C01378=1093.249,362.151,-91.490,178.091,22.265,153.224
C01379=1093.255,362.398,-91.525,178.094,22.270,153.224
C01380=1093.261,362.645,-91.561,178.097,22.274,153.225
C01381=1093.266,362.892,-91.596,178.100,22.279,153.226
C01382=1093.273,363.140,-91.632,178.103,22.284,153.226
C01383=1093.279,363.387,-91.667,178.105,22.289,153.227
C01384=1093.285,363.634,-91.703,178.108,22.294,153.228
C01385=1093.291,363.882,-91.738,178.112,22.299,153.229
C01386=1093.296,364.129,-91.774,178.115,22.304,153.229
C01387=1093.302,364.377,-91.810,178.118,22.309,153.230
C01388=1093.308,364.624,-91.845,178.121,22.313,153.231
C01389=1093.314,364.871,-91.881,178.124,22.318,153.231
C01390=1093.320,365.118,-91.917,178.127,22.324,153.232
C01391=1093.326,365.366,-91.953,178.130,22.329,153.233
C01392=1093.331,365.613,-91.988,178.133,22.333,153.234
C01393=1093.337,365.861,-92.024,178.136,22.339,153.235
C01394=1093.343,366.108,-92.060,178.139,22.344,153.235
C01395=1093.349,366.355,-92.095,178.142,22.349,153.236
C01396=1093.355,366.602,-92.131,178.145,22.354,153.237
C01397=1093.360,366.850,-92.168,178.147,22.359,153.238
C01398=1093.366,367.097,-92.203,178.151,22.364,153.238
C01399=1093.372,367.345,-92.239,178.154,22.369,153.239
C01400=1093.378,367.592,-92.275,178.157,22.375,153.240
C01401=1093.384,367.839,-92.311,178.160,22.380,153.241
C01402=1093.390,368.087,-92.346,178.162,22.385,153.241
C01403=1093.395,368.334,-92.383,178.165,22.390,153.242
C01404=1093.401,368.581,-92.419,178.169,22.395,153.243
C01405=1093.407,368.828,-92.455,178.172,22.400,153.244
C01406=1093.413,369.076,-92.491,178.175,22.406,153.245
C01407=1093.419,369.323,-92.526,178.178,22.411,153.245
C01408=1093.424,369.570,-92.563,178.180,22.416,153.246
C01409=1093.434,369.971,-92.621,178.185,22.425,153.248
C01410=1093.443,370.370,-92.680,178.190,22.433,153.249
C01411=1093.453,370.772,-92.738,178.195,22.442,153.250
C01412=1093.462,371.172,-92.798,178.200,22.451,153.252
C01413=1093.468,371.420,-92.833,178.203,22.456,153.252
C01414=1093.475,371.667,-92.870,178.206,22.461,153.253
C01415=1093.480,371.913,-92.906,178.209,22.467,153.254
C01416=1093.486,372.161,-92.942,178.212,22.472,153.255
C01417=1093.492,372.408,-92.979,178.215,22.477,153.256
C01418=1093.498,372.655,-93.015,178.218,22.483,153.257
C01419=1093.504,372.903,-93.051,178.221,22.488,153.257
C01420=1093.510,373.150,-93.088,178.224,22.494,153.258
C01421=1093.516,373.397,-93.124,178.227,22.499,153.259
C01422=1093.521,373.645,-93.160,178.230,22.504,153.260
C01423=1093.527,373.892,-93.197,178.233,22.509,153.261
C01424=1093.534,374.139,-93.233,178.236,22.515,153.262
C01425=1093.539,374.386,-93.270,178.239,22.520,153.263
C01426=1093.546,374.633,-93.307,178.242,22.526,153.263
C01427=1093.551,374.881,-93.343,178.245,22.532,153.264
C01428=1093.557,375.127,-93.379,178.248,22.538,153.265
C01429=1093.562,375.375,-93.416,178.251,22.543,153.266
C01430=1093.569,375.622,-93.452,178.254,22.549,153.267
C01431=1093.574,375.869,-93.490,178.257,22.555,153.268
C01432=1093.580,376.116,-93.526,178.260,22.560,153.269
C01433=1093.586,376.364,-93.563,178.263,22.566,153.270
C01434=1093.592,376.610,-93.599,178.266,22.572,153.271
C01435=1093.597,376.857,-93.636,178.269,22.577,153.272
C01436=1093.604,377.104,-93.673,178.271,22.582,153.273
C01437=1093.609,377.352,-93.710,178.274,22.588,153.274
C01438=1093.615,377.599,-93.747,178.277,22.594,153.274
C01439=1093.621,377.846,-93.783,178.280,22.600,153.275
C01440=1093.627,378.094,-93.820,178.283,22.605,153.276
C01441=1093.633,378.341,-93.857,178.286,22.611,153.277
C01442=1093.639,378.588,-93.894,178.289,22.617,153.278
C01443=1093.644,378.835,-93.931,178.292,22.623,153.279
C01444=1093.651,379.082,-93.967,178.295,22.628,153.280
C01445=1093.657,379.329,-94.005,178.298,22.634,153.281
C01446=1093.663,379.576,-94.041,178.300,22.640,153.282
C01447=1093.669,379.824,-94.078,178.304,22.646,153.283
C01448=1093.674,380.071,-94.115,178.306,22.652,153.284
C01449=1093.680,380.318,-94.152,178.309,22.657,153.285
C01450=1093.686,380.565,-94.190,178.312,22.663,153.286
C01451=1093.692,380.812,-94.227,178.315,22.669,153.287
C01452=1093.698,381.059,-94.263,178.318,22.675,153.288
C01453=1093.704,381.306,-94.301,178.321,22.681,153.289
C01454=1093.710,381.553,-94.338,178.324,22.687,153.290
C01455=1093.716,381.800,-94.374,178.327,22.693,153.291
C01456=1093.722,382.047,-94.412,178.330,22.699,153.292
C01457=1093.728,382.294,-94.449,178.333,22.705,153.293
C01458=1093.734,382.541,-94.486,178.336,22.711,153.294
C01459=1093.740,382.788,-94.523,178.339,22.717,153.295
C01460=1093.746,383.036,-94.560,178.342,22.723,153.296
C01461=1093.755,383.422,-94.619,178.346,22.732,153.298
C01462=1093.764,383.807,-94.677,178.351,22.742,153.299
C01463=1093.773,384.194,-94.736,178.355,22.751,153.301
C01464=1093.782,384.580,-94.795,178.360,22.761,153.303
C01465=1093.788,384.827,-94.832,178.363,22.767,153.304
C01466=1093.794,385.074,-94.869,178.366,22.773,153.305
C01467=1093.800,385.320,-94.907,178.369,22.780,153.306
C01468=1093.806,385.568,-94.944,178.372,22.786,153.307
C01469=1093.812,385.814,-94.982,178.375,22.793,153.308
C01470=1093.818,386.061,-95.019,178.378,22.798,153.309
C01471=1093.823,386.309,-95.056,178.381,22.805,153.310
C01472=1093.829,386.555,-95.094,178.383,22.811,153.311
C01473=1093.836,386.845,-95.138,178.387,22.819,153.313
C01474=1093.843,387.133,-95.183,178.390,22.826,153.314
C01475=1093.850,387.422,-95.226,178.394,22.833,153.315
C01476=1093.857,387.711,-95.270,178.397,22.840,153.316
C01477=1093.863,387.958,-95.308,178.400,22.847,153.317
C01478=1093.869,388.205,-95.345,178.403,22.853,153.319
C01479=1093.875,388.453,-95.384,178.406,22.860,153.320
C01480=1093.881,388.699,-95.422,178.409,22.866,153.321
C01481=1093.886,388.946,-95.460,178.412,22.873,153.322
C01482=1093.892,389.193,-95.497,178.414,22.879,153.323
C01483=1093.899,389.440,-95.536,178.417,22.886,153.324
C01484=1093.905,389.687,-95.573,178.420,22.892,153.325
C01485=1093.911,389.934,-95.611,178.424,22.899,153.327
C01486=1093.917,390.180,-95.649,178.426,22.905,153.328
C01487=1093.923,390.428,-95.687,178.429,22.912,153.329
C01488=1093.929,390.675,-95.725,178.432,22.918,153.330
C01489=1093.935,390.921,-95.762,178.435,22.924,153.331
C01490=1093.941,391.168,-95.800,178.438,22.932,153.332
C01491=1093.947,391.416,-95.838,178.441,22.938,153.334
C01492=1093.952,391.663,-95.877,178.444,22.944,153.335
C01493=1093.959,391.910,-95.915,178.446,22.951,153.336
C01494=1093.965,392.157,-95.953,178.449,22.957,153.337
C01495=1093.971,392.404,-95.990,178.453,22.965,153.338
C01496=1093.977,392.651,-96.028,178.455,22.971,153.340
C01497=1093.983,392.897,-96.068,178.458,22.978,153.341
C01498=1093.989,393.144,-96.105,178.461,22.984,153.342
C01499=1093.995,393.391,-96.143,178.464,22.992,153.343
C01500=1094.000,393.639,-96.182,178.467,22.998,153.345
C01501=1094.007,393.885,-96.220,178.469,23.005,153.346
C01502=1094.013,394.132,-96.258,178.472,23.012,153.347
C01503=1094.018,394.379,-96.297,178.476,23.019,153.348
C01504=1094.024,394.625,-96.335,178.478,23.026,153.349
C01505=1094.031,394.873,-96.373,178.481,23.032,153.351
C01506=1094.036,395.120,-96.412,178.483,23.039,153.352
C01507=1094.043,395.367,-96.450,178.487,23.046,153.353
C01508=1094.049,395.614,-96.488,178.490,23.053,153.355
C01509=1094.054,395.861,-96.527,178.492,23.060,153.356
C01510=1094.061,396.107,-96.565,178.496,23.067,153.357
C01511=1094.066,396.354,-96.604,178.498,23.075,153.359
C01512=1094.073,396.601,-96.643,178.501,23.081,153.360
C01513=1094.077,396.821,-96.677,178.504,23.088,153.361
C01514=1094.083,397.042,-96.712,178.506,23.094,153.362
C01515=1094.088,397.263,-96.746,178.508,23.100,153.363
C01516=1094.094,397.483,-96.781,178.511,23.107,153.365
C01517=1094.099,397.703,-96.815,178.514,23.113,153.366
C01518=1094.105,397.924,-96.849,178.516,23.120,153.367
C01519=1094.109,398.144,-96.884,178.518,23.126,153.368
C01520=1094.115,398.365,-96.919,178.521,23.132,153.369
C01521=1094.121,398.612,-96.957,178.524,23.139,153.371
C01522=1094.127,398.859,-96.996,178.527,23.147,153.372
C01523=1094.133,399.105,-97.035,178.530,23.154,153.373
C01524=1094.139,399.353,-97.073,178.533,23.161,153.375
C01525=1094.145,399.600,-97.113,178.535,23.169,153.376
C01526=1094.151,399.846,-97.151,178.538,23.175,153.377
C01527=1094.157,400.094,-97.190,178.541,23.183,153.379
C01528=1094.163,400.340,-97.229,178.544,23.190,153.380
C01529=1094.169,400.587,-97.268,178.546,23.198,153.382
C01530=1094.175,400.833,-97.307,178.550,23.205,153.383
C01531=1094.181,401.081,-97.346,178.552,23.213,153.384
C01532=1094.187,401.328,-97.385,178.556,23.220,153.386
C01533=1094.193,401.574,-97.424,178.558,23.228,153.387
C01534=1094.199,401.822,-97.463,178.561,23.236,153.389
C01535=1094.204,402.068,-97.502,178.564,23.243,153.390
C01536=1094.211,402.315,-97.541,178.566,23.250,153.392
C01537=1094.217,402.562,-97.580,178.569,23.258,153.393
C01538=1094.223,402.808,-97.619,178.572,23.265,153.395
C01539=1094.229,403.056,-97.659,178.575,23.273,153.396
C01540=1094.235,403.303,-97.698,178.578,23.281,153.397
C01541=1094.241,403.549,-97.737,178.581,23.288,153.399
C01542=1094.247,403.796,-97.776,178.583,23.296,153.400
C01543=1094.253,404.043,-97.816,178.587,23.304,153.402
C01544=1094.259,404.290,-97.855,178.589,23.311,153.403
C01545=1094.265,404.537,-97.894,178.592,23.319,153.405
C01546=1094.271,404.784,-97.933,178.595,23.327,153.406
C01547=1094.278,405.031,-97.972,178.598,23.335,153.408
C01548=1094.284,405.276,-98.012,178.600,23.342,153.409
C01549=1094.290,405.524,-98.052,178.604,23.350,153.411
C01550=1094.296,405.771,-98.091,178.606,23.358,153.412
C01551=1094.302,406.018,-98.130,178.609,23.366,153.414
C01552=1094.308,406.264,-98.170,178.611,23.374,153.416
C01553=1094.314,406.511,-98.210,178.615,23.382,153.417
C01554=1094.320,406.758,-98.249,178.618,23.390,153.419
C01555=1094.326,407.005,-98.288,178.620,23.398,153.420
C01556=1094.332,407.251,-98.328,178.623,23.406,153.422
C01557=1094.338,407.498,-98.368,178.626,23.414,153.423
C01558=1094.344,407.745,-98.407,178.629,23.422,153.425
C01559=1094.350,407.992,-98.447,178.632,23.430,153.427
C01560=1094.356,408.239,-98.487,178.634,23.438,153.428
C01561=1094.362,408.485,-98.526,178.637,23.447,153.430
C01562=1094.367,408.732,-98.567,178.641,23.455,153.431
C01563=1094.374,408.979,-98.607,178.643,23.463,153.433
C01564=1094.380,409.226,-98.646,178.646,23.472,153.435
C01565=1094.386,409.472,-98.686,178.648,23.480,153.436
C01566=1094.392,409.719,-98.725,178.651,23.488,153.438
C01567=1094.398,409.965,-98.765,178.654,23.496,153.440
C01568=1094.403,410.213,-98.805,178.657,23.504,153.441
C01569=1094.409,410.434,-98.842,178.660,23.512,153.443
C01570=1094.414,410.654,-98.877,178.662,23.520,153.444
C01571=1094.420,410.875,-98.913,178.665,23.527,153.446
C01572=1094.425,411.096,-98.949,178.667,23.535,153.447
C01573=1094.431,411.317,-98.985,178.670,23.543,153.449
C01574=1094.436,411.537,-99.021,178.672,23.550,153.450
C01575=1094.441,411.758,-99.056,178.674,23.558,153.452
C01576=1094.447,411.979,-99.092,178.677,23.565,153.453
C01577=1094.453,412.225,-99.132,178.680,23.574,153.455
C01578=1094.459,412.472,-99.172,178.683,23.582,153.457
C01579=1094.465,412.719,-99.213,178.686,23.591,153.459
C01580=1094.471,412.966,-99.252,178.688,23.599,153.460
C01581=1094.477,413.212,-99.293,178.691,23.608,153.462
C01582=1094.484,413.459,-99.333,178.694,23.617,153.464
C01583=1094.489,413.706,-99.373,178.697,23.626,153.465
C01584=1094.496,413.952,-99.414,178.700,23.635,153.467
C01585=1094.502,414.199,-99.454,178.702,23.643,153.469
C01586=1094.508,414.445,-99.494,178.706,23.652,153.471
C01587=1094.514,414.692,-99.535,178.709,23.661,153.473
C01588=1094.521,414.938,-99.575,178.712,23.670,153.474
C01589=1094.526,415.185,-99.615,178.715,23.678,153.476
C01590=1094.533,415.432,-99.656,178.718,23.687,153.478
C01591=1094.539,415.678,-99.696,178.720,23.696,153.480
C01592=1094.545,415.925,-99.737,178.722,23.705,153.482
C01593=1094.551,416.172,-99.777,178.725,23.714,153.483
C01594=1094.558,416.419,-99.817,178.728,23.723,153.485
C01595=1094.564,416.666,-99.858,178.731,23.732,153.487
C01596=1094.570,416.912,-99.899,178.734,23.741,153.489
C01597=1094.576,417.158,-99.940,178.737,23.751,153.491
C01598=1094.582,417.405,-99.980,178.740,23.760,153.493
C01599=1094.588,417.652,-100.020,178.743,23.769,153.495
C01600=1094.594,417.898,-100.062,178.746,23.778,153.497
C01601=1094.600,418.144,-100.102,178.749,23.788,153.498
C01602=1094.606,418.391,-100.143,178.751,23.797,153.500
C01603=1094.612,418.638,-100.184,178.754,23.806,153.502
C01604=1094.618,418.884,-100.224,178.756,23.815,153.504
C01605=1094.624,419.131,-100.265,178.759,23.825,153.506
C01606=1094.631,419.377,-100.306,178.762,23.834,153.508
C01607=1094.637,419.624,-100.347,178.765,23.843,153.510
C01608=1094.643,419.870,-100.389,178.768,23.853,153.512
C01609=1094.649,420.117,-100.429,178.771,23.862,153.514
C01610=1094.655,420.363,-100.470,178.774,23.872,153.516
C01611=1094.661,420.610,-100.511,178.776,23.882,153.518
C01612=1094.668,420.857,-100.552,178.779,23.891,153.520
C01613=1094.674,421.103,-100.593,178.782,23.901,153.522
C01614=1094.680,421.350,-100.634,178.786,23.910,153.524
C01615=1094.686,421.596,-100.675,178.788,23.920,153.526
C01616=1094.693,421.843,-100.716,178.791,23.930,153.528
C01617=1094.699,422.089,-100.758,178.794,23.940,153.530
C01618=1094.704,422.335,-100.799,178.797,23.949,153.532
C01619=1094.711,422.582,-100.839,178.800,23.959,153.534
C01620=1094.717,422.829,-100.881,178.802,23.969,153.536
C01621=1094.723,423.075,-100.923,178.805,23.979,153.538
C01622=1094.729,423.321,-100.964,178.808,23.989,153.540
C01623=1094.735,423.568,-101.005,178.810,23.998,153.542
C01624=1094.741,423.815,-101.047,178.814,24.009,153.544
C01625=1094.747,424.042,-101.084,178.816,24.018,153.546
C01626=1094.753,424.270,-101.124,178.819,24.027,153.548
C01627=1094.759,424.498,-101.162,178.822,24.037,153.550
C01628=1094.764,424.726,-101.200,178.824,24.046,153.552
C01629=1094.770,424.954,-101.238,178.827,24.056,153.554
C01630=1094.776,425.182,-101.276,178.830,24.065,153.556
C01631=1094.781,425.411,-101.315,178.831,24.074,153.558
C01632=1094.787,425.638,-101.354,178.834,24.084,153.560
C01633=1094.794,425.884,-101.395,178.837,24.094,153.562
C01634=1094.800,426.131,-101.437,178.840,24.105,153.565
C01635=1094.806,426.377,-101.478,178.843,24.115,153.567
C01636=1094.812,426.624,-101.520,178.846,24.125,153.569
C01637=1094.818,426.870,-101.561,178.848,24.135,153.571
C01638=1094.825,427.117,-101.603,178.852,24.146,153.573
C01639=1094.831,427.363,-101.645,178.854,24.156,153.576
C01640=1094.838,427.609,-101.687,178.857,24.167,153.578
C01641=1094.844,427.855,-101.729,178.860,24.177,153.580
C01642=1094.850,428.102,-101.770,178.863,24.188,153.583
C01643=1094.856,428.349,-101.812,178.866,24.198,153.585
C01644=1094.862,428.594,-101.855,178.868,24.209,153.587
C01645=1094.868,428.841,-101.897,178.871,24.220,153.589
C01646=1094.874,429.088,-101.938,178.874,24.231,153.592
C01647=1094.881,429.334,-101.981,178.877,24.241,153.594
C01648=1094.887,429.580,-102.022,178.879,24.252,153.596
C01649=1094.894,429.826,-102.065,178.883,24.263,153.599
C01650=1094.899,430.073,-102.107,178.885,24.274,153.601
C01651=1094.906,430.319,-102.149,178.888,24.285,153.603
C01652=1094.912,430.565,-102.191,178.891,24.296,153.606
C01653=1094.919,430.812,-102.233,178.894,24.307,153.608
C01654=1094.925,431.058,-102.275,178.897,24.318,153.611
C01655=1094.931,431.304,-102.318,178.899,24.329,153.613
C01656=1094.937,431.550,-102.360,178.902,24.340,153.615
C01657=1094.943,431.797,-102.402,178.905,24.351,153.618
C01658=1094.950,432.042,-102.444,178.908,24.362,153.620
C01659=1094.956,432.289,-102.487,178.911,24.374,153.623
C01660=1094.962,432.535,-102.528,178.913,24.385,153.625
C01661=1094.969,432.782,-102.571,178.916,24.396,153.628
C01662=1094.974,433.027,-102.614,178.919,24.408,153.630
C01663=1094.981,433.274,-102.656,178.922,24.419,153.632
C01664=1094.987,433.520,-102.699,178.925,24.430,153.635
C01665=1094.993,433.767,-102.741,178.927,24.442,153.638
C01666=1095.000,434.013,-102.783,178.930,24.454,153.640
C01667=1095.005,434.259,-102.826,178.933,24.465,153.643
C01668=1095.012,434.505,-102.869,178.936,24.477,153.645
C01669=1095.018,434.751,-102.912,178.938,24.488,153.648
C01670=1095.025,434.997,-102.954,178.942,24.500,153.650
C01671=1095.031,435.244,-102.997,178.944,24.512,153.653
C01672=1095.036,435.490,-103.040,178.947,24.524,153.656
C01673=1095.043,435.736,-103.083,178.949,24.535,153.658
C01674=1095.049,435.983,-103.126,178.952,24.547,153.661
C01675=1095.056,436.228,-103.169,178.956,24.559,153.663
C01676=1095.062,436.474,-103.212,178.958,24.571,153.666
C01677=1095.069,436.720,-103.254,178.961,24.583,153.669
C01678=1095.074,436.966,-103.297,178.963,24.595,153.671
C01679=1095.081,437.213,-103.340,178.967,24.607,153.674
C01680=1095.088,437.459,-103.383,178.970,24.619,153.677
C01681=1095.094,437.699,-103.425,178.972,24.631,153.679
C01682=1095.099,437.939,-103.467,178.974,24.643,153.682
C01683=1095.106,438.179,-103.509,178.978,24.655,153.685
C01684=1095.113,438.420,-103.551,178.980,24.667,153.687
C01685=1095.118,438.661,-103.593,178.983,24.679,153.690
C01686=1095.125,438.901,-103.636,178.985,24.691,153.693
C01687=1095.131,439.141,-103.678,178.988,24.703,153.695
C01688=1095.137,439.382,-103.720,178.991,24.715,153.698
C01689=1095.144,439.628,-103.762,178.994,24.728,153.701
C01690=1095.150,439.874,-103.806,178.997,24.740,153.704
C01691=1095.156,440.121,-103.849,179.000,24.753,153.706
C01692=1095.163,440.367,-103.893,179.002,24.765,153.709
C01693=1095.169,440.612,-103.936,179.005,24.778,153.712
C01694=1095.175,440.858,-103.979,179.008,24.791,153.715
C01695=1095.182,441.104,-104.023,179.010,24.803,153.718
C01696=1095.188,441.350,-104.067,179.013,24.816,153.721
C01697=1095.194,441.597,-104.110,179.016,24.830,153.724
C01698=1095.201,441.842,-104.153,179.019,24.842,153.727
C01699=1095.207,442.088,-104.197,179.022,24.855,153.730
C01700=1095.214,442.334,-104.241,179.024,24.868,153.732
C01701=1095.220,442.580,-104.284,179.027,24.881,153.735
C01702=1095.226,442.826,-104.328,179.030,24.895,153.738
C01703=1095.233,443.072,-104.372,179.033,24.908,153.741
C01704=1095.239,443.318,-104.415,179.036,24.921,153.744
C01705=1095.246,443.564,-104.459,179.038,24.934,153.747
C01706=1095.252,443.810,-104.503,179.041,24.948,153.750
C01707=1095.259,444.056,-104.547,179.044,24.961,153.754
C01708=1095.265,444.302,-104.591,179.047,24.975,153.757
C01709=1095.271,444.548,-104.635,179.049,24.988,153.760
C01710=1095.278,444.794,-104.679,179.051,25.001,153.763
C01711=1095.284,445.040,-104.722,179.053,25.014,153.766
C01712=1095.291,445.286,-104.766,179.054,25.028,153.769
C01713=1095.297,445.531,-104.811,179.056,25.041,153.772
C01714=1095.304,445.777,-104.855,179.058,25.054,153.775
C01715=1095.310,446.023,-104.898,179.059,25.067,153.779
C01716=1095.317,446.269,-104.942,179.060,25.080,153.782
C01717=1095.322,446.516,-104.987,179.061,25.094,153.785
C01718=1095.329,446.761,-105.031,179.062,25.107,153.788
C01719=1095.336,447.007,-105.075,179.063,25.120,153.791
C01720=1095.342,447.253,-105.119,179.064,25.133,153.795
C01721=1095.348,447.499,-105.163,179.064,25.147,153.798
C01722=1095.354,447.745,-105.208,179.064,25.160,153.801
C01723=1095.361,447.991,-105.252,179.065,25.173,153.805
C01724=1095.368,448.237,-105.296,179.065,25.186,153.808
C01725=1095.375,448.483,-105.341,179.065,25.200,153.811
C01726=1095.381,448.729,-105.385,179.064,25.212,153.815
C01727=1095.387,448.974,-105.430,179.064,25.225,153.818
C01728=1095.393,449.220,-105.474,179.064,25.239,153.821
C01729=1095.400,449.466,-105.517,179.063,25.251,153.825
C01730=1095.407,449.712,-105.562,179.062,25.265,153.828
C01731=1095.413,449.957,-105.607,179.061,25.277,153.832
C01732=1095.421,450.203,-105.650,179.060,25.290,153.835
C01733=1095.031,450.195,-105.819,179.006,25.499,153.895
C01734=1095.022,449.948,-105.774,179.006,25.488,153.891
C01735=1095.016,449.702,-105.730,179.007,25.474,153.888
C01736=1095.010,449.457,-105.685,179.008,25.461,153.885
C01737=1095.003,449.211,-105.640,179.009,25.448,153.881
C01738=1094.997,448.965,-105.597,179.009,25.435,153.878
C01739=1094.990,448.720,-105.552,179.009,25.422,153.874
C01740=1094.983,448.474,-105.508,179.010,25.409,153.871
C01741=1094.977,448.228,-105.463,179.010,25.396,153.868
C01742=1094.970,447.982,-105.419,179.010,25.383,153.864
C01743=1094.964,447.736,-105.374,179.010,25.369,153.861
C01744=1094.957,447.490,-105.330,179.009,25.356,153.858
C01745=1094.952,447.244,-105.286,179.008,25.343,153.854
C01746=1094.945,446.999,-105.241,179.008,25.329,153.851
C01747=1094.938,446.753,-105.198,179.006,25.316,153.848
C01748=1094.932,446.507,-105.154,179.005,25.302,153.845
C01749=1094.925,446.261,-105.109,179.004,25.289,153.841
C01750=1094.919,446.014,-105.064,179.003,25.276,153.838
C01751=1094.913,445.768,-105.021,179.002,25.263,153.835
C01752=1094.906,445.522,-104.977,179.000,25.249,153.832
C01753=1094.899,445.277,-104.932,178.998,25.236,153.829
C01754=1094.893,445.031,-104.888,178.997,25.223,153.825
C01755=1094.887,444.785,-104.844,178.994,25.209,153.822
C01756=1094.880,444.539,-104.801,178.992,25.196,153.819
C01757=1094.874,444.293,-104.757,178.990,25.183,153.816
C01758=1094.867,444.047,-104.713,178.987,25.169,153.813
C01759=1094.861,443.801,-104.669,178.984,25.156,153.810
C01760=1094.854,443.555,-104.625,178.981,25.142,153.807
C01761=1094.848,443.309,-104.581,178.979,25.129,153.804
C01762=1094.842,443.063,-104.537,178.976,25.116,153.801
C01763=1094.835,442.817,-104.494,178.973,25.102,153.798
C01764=1094.829,442.571,-104.450,178.970,25.089,153.795
C01765=1094.822,442.325,-104.406,178.967,25.076,153.792
C01766=1094.816,442.079,-104.362,178.965,25.063,153.789
C01767=1094.810,441.833,-104.318,178.962,25.050,153.786
C01768=1094.804,441.588,-104.275,178.959,25.037,153.783
C01769=1094.797,441.342,-104.231,178.956,25.024,153.780
C01770=1094.790,441.096,-104.188,178.953,25.011,153.777
C01771=1094.784,440.850,-104.144,178.950,24.998,153.774
C01772=1094.778,440.604,-104.101,178.947,24.985,153.772
C01773=1094.771,440.357,-104.057,178.944,24.973,153.769
C01774=1094.764,440.112,-104.014,178.942,24.960,153.766
C01775=1094.758,439.866,-103.970,178.939,24.947,153.763
C01776=1094.752,439.620,-103.928,178.936,24.935,153.760
C01777=1094.746,439.374,-103.884,178.933,24.922,153.757
C01778=1094.739,439.138,-103.842,178.930,24.910,153.755
C01779=1094.733,438.903,-103.802,178.928,24.899,153.752
C01780=1094.728,438.668,-103.760,178.925,24.887,153.749
C01781=1094.721,438.432,-103.719,178.922,24.875,153.747
C01782=1094.714,438.197,-103.677,178.919,24.863,153.744
C01783=1094.708,437.962,-103.636,178.916,24.851,153.742
C01784=1094.703,437.727,-103.595,178.914,24.839,153.739
C01785=1094.697,437.492,-103.554,178.911,24.828,153.736
C01786=1094.691,437.245,-103.511,178.908,24.815,153.734
C01787=1094.683,436.999,-103.468,178.906,24.804,153.731
C01788=1094.677,436.753,-103.425,178.902,24.791,153.728
C01789=1094.671,436.507,-103.382,178.900,24.779,153.726
C01790=1094.665,436.261,-103.339,178.897,24.768,153.723
C01791=1094.658,436.015,-103.296,178.894,24.755,153.720
C01792=1094.652,435.769,-103.253,178.891,24.743,153.718
C01793=1094.646,435.523,-103.210,178.888,24.732,153.715
C01794=1094.639,435.276,-103.168,178.886,24.720,153.712
C01795=1094.634,435.030,-103.125,178.882,24.708,153.710
C01796=1094.627,434.784,-103.082,178.880,24.696,153.707
C01797=1094.621,434.537,-103.039,178.877,24.684,153.705
C01798=1094.615,434.292,-102.997,178.874,24.673,153.702
C01799=1094.608,434.045,-102.954,178.871,24.661,153.700
C01800=1094.602,433.800,-102.912,178.868,24.649,153.697
C01801=1094.596,433.553,-102.868,178.865,24.638,153.694
C01802=1094.589,433.307,-102.826,178.863,24.627,153.692
C01803=1094.584,433.061,-102.783,178.859,24.615,153.689
C01804=1094.577,432.815,-102.741,178.857,24.604,153.687
C01805=1094.571,432.569,-102.698,178.854,24.592,153.685
C01806=1094.565,432.322,-102.656,178.851,24.581,153.682
C01807=1094.558,432.076,-102.614,178.848,24.570,153.680
C01808=1094.552,431.830,-102.571,178.845,24.558,153.677
C01809=1094.545,431.584,-102.529,178.843,24.547,153.675
C01810=1094.540,431.337,-102.487,178.839,24.536,153.672
C01811=1094.533,431.091,-102.444,178.837,24.525,153.670
C01812=1094.526,430.845,-102.402,178.834,24.514,153.668
